MoveJ RelTool (starting_position, 124, 300, -195 \Rx:=-0.5, \Ry:=-1.8, \Rz:=0), v200, z200, Tooldata_7;
MoveJ RelTool (starting_position, 124, 300, -195 \Rx:=-0.2, \Ry:=-1.8, \Rz:=0), v200, z200, Tooldata_7;
MoveJ RelTool (starting_position, 124, 300, -195 \Rx:=0.2, \Ry:=-1.8, \Rz:=0), v200, z200, Tooldata_7;
MoveJ RelTool (starting_position, 125, 300, -194 \Rx:=0.6, \Ry:=-1.5, \Rz:=0), v200, z200, Tooldata_7;
MoveJ RelTool (starting_position, 125, 300, -194 \Rx:=1, \Ry:=-1.5, \Rz:=0), v200, z200, Tooldata_7;
MoveJ RelTool (starting_position, 126, 300, -193 \Rx:=1.5, \Ry:=-1.5, \Rz:=0), v200, z200, Tooldata_7;
MoveJ RelTool (starting_position, 127, 300, -193 \Rx:=2, \Ry:=-1.2, \Rz:=0), v200, z200, Tooldata_7;
MoveJ RelTool (starting_position, 128, 300, -192 \Rx:=2.5, \Ry:=-0.9, \Rz:=0), v200, z200, Tooldata_7;
MoveJ RelTool (starting_position, 130, 300, -192 \Rx:=3, \Ry:=-0.9, \Rz:=0), v200, z200, Tooldata_7;
MoveJ RelTool (starting_position, 132, 300, -191 \Rx:=3.4, \Ry:=-0.3, \Rz:=0), v200, z200, Tooldata_7;
MoveJ RelTool (starting_position, 134, 300, -191 \Rx:=3.9, \Ry:=0, \Rz:=0), v200, z200, Tooldata_7;
MoveJ RelTool (starting_position, 136, 300, -191 \Rx:=4.3, \Ry:=0.3, \Rz:=0), v200, z200, Tooldata_7;
MoveJ RelTool (starting_position, 138, 300, -190 \Rx:=4.6, \Ry:=0.6, \Rz:=0), v200, z200, Tooldata_7;
MoveJ RelTool (starting_position, 140, 300, -190 \Rx:=5, \Ry:=1.2, \Rz:=0), v200, z200, Tooldata_7;
MoveJ RelTool (starting_position, 143, 300, -189 \Rx:=5.3, \Ry:=1.5, \Rz:=0), v200, z200, Tooldata_7;
MoveJ RelTool (starting_position, 145, 300, -189 \Rx:=5.5, \Ry:=2.1, \Rz:=0), v200, z200, Tooldata_7;
MoveJ RelTool (starting_position, 148, 300, -189 \Rx:=5.7, \Ry:=2.4, \Rz:=0), v200, z200, Tooldata_7;
MoveJ RelTool (starting_position, 151, 300, -189 \Rx:=5.9, \Ry:=3, \Rz:=0), v200, z200, Tooldata_7;
MoveJ RelTool (starting_position, 155, 300, -189 \Rx:=6, \Ry:=3.6, \Rz:=0), v200, z200, Tooldata_7;
MoveJ RelTool (starting_position, 158, 300, -189 \Rx:=6.1, \Ry:=4.2, \Rz:=0), v200, z200, Tooldata_7;
MoveJ RelTool (starting_position, 162, 300, -189 \Rx:=6, \Ry:=4.8, \Rz:=0), v200, z200, Tooldata_7;
MoveJ RelTool (starting_position, 166, 300, -190 \Rx:=6, \Ry:=5.4, \Rz:=0), v200, z200, Tooldata_7;
MoveJ RelTool (starting_position, 170, 300, -190 \Rx:=5.9, \Ry:=6.3, \Rz:=0), v200, z200, Tooldata_7;
MoveJ RelTool (starting_position, 174, 300, -191 \Rx:=5.8, \Ry:=6.9, \Rz:=0), v200, z200, Tooldata_7;
MoveJ RelTool (starting_position, 178, 300, -191 \Rx:=5.7, \Ry:=7.8, \Rz:=0), v200, z200, Tooldata_7;
MoveJ RelTool (starting_position, 182, 300, -192 \Rx:=5.6, \Ry:=8.4, \Rz:=0), v200, z200, Tooldata_7;
MoveJ RelTool (starting_position, 186, 300, -193 \Rx:=5.5, \Ry:=9, \Rz:=0), v200, z200, Tooldata_7;
MoveJ RelTool (starting_position, 189, 300, -194 \Rx:=5.3, \Ry:=9.6, \Rz:=0), v200, z200, Tooldata_7;
MoveJ RelTool (starting_position, 193, 300, -195 \Rx:=5.3, \Ry:=10.5, \Rz:=0), v200, z200, Tooldata_7;
MoveJ RelTool (starting_position, 197, 300, -196 \Rx:=5.2, \Ry:=10.8, \Rz:=0), v200, z200, Tooldata_7;
MoveJ RelTool (starting_position, 200, 300, -197 \Rx:=5.2, \Ry:=11.7, \Rz:=0), v200, z200, Tooldata_7;
MoveJ RelTool (starting_position, 204, 300, -198 \Rx:=5.2, \Ry:=12.3, \Rz:=0), v200, z200, Tooldata_7;
MoveJ RelTool (starting_position, 207, 300, -199 \Rx:=5.3, \Ry:=12.6, \Rz:=0), v200, z200, Tooldata_7;
MoveJ RelTool (starting_position, 211, 300, -200 \Rx:=5.4, \Ry:=13.2, \Rz:=0), v200, z200, Tooldata_7;
MoveJ RelTool (starting_position, 214, 300, -202 \Rx:=5.5, \Ry:=14.1, \Rz:=0), v200, z200, Tooldata_7;
MoveJ RelTool (starting_position, 218, 300, -203 \Rx:=5.8, \Ry:=14.7, \Rz:=0), v200, z200, Tooldata_7;
MoveJ RelTool (starting_position, 221, 300, -205 \Rx:=5.9, \Ry:=15.3, \Rz:=0), v200, z200, Tooldata_7;
MoveJ RelTool (starting_position, 224, 300, -206 \Rx:=6.1, \Ry:=15.6, \Rz:=0), v200, z200, Tooldata_7;
MoveJ RelTool (starting_position, 227, 300, -208 \Rx:=6.4, \Ry:=16.2, \Rz:=0), v200, z200, Tooldata_7;
MoveJ RelTool (starting_position, 229, 300, -210 \Rx:=6.8, \Ry:=16.5, \Rz:=0), v200, z200, Tooldata_7;
MoveJ RelTool (starting_position, 231, 300, -212 \Rx:=7.2, \Ry:=17.1, \Rz:=0), v200, z200, Tooldata_7;
MoveJ RelTool (starting_position, 233, 300, -214 \Rx:=7.6, \Ry:=17.4, \Rz:=0), v200, z200, Tooldata_7;
MoveJ RelTool (starting_position, 235, 300, -216 \Rx:=8.1, \Ry:=17.7, \Rz:=0), v200, z200, Tooldata_7;
MoveJ RelTool (starting_position, 237, 300, -218 \Rx:=8.5, \Ry:=18, \Rz:=0), v200, z200, Tooldata_7;
MoveJ RelTool (starting_position, 238, 300, -221 \Rx:=8.9, \Ry:=18, \Rz:=0), v200, z200, Tooldata_7;
MoveJ RelTool (starting_position, 238, 300, -223 \Rx:=9.3, \Ry:=18.3, \Rz:=0), v200, z200, Tooldata_7;
MoveJ RelTool (starting_position, 238, 300, -226 \Rx:=9.8, \Ry:=18.3, \Rz:=0), v200, z200, Tooldata_7;
MoveJ RelTool (starting_position, 238, 300, -228 \Rx:=10.2, \Ry:=18.3, \Rz:=0), v200, z200, Tooldata_7;
MoveJ RelTool (starting_position, 238, 300, -231 \Rx:=10.5, \Ry:=18, \Rz:=0), v200, z200, Tooldata_7;
MoveJ RelTool (starting_position, 237, 300, -234 \Rx:=10.9, \Ry:=18, \Rz:=0), v200, z200, Tooldata_7;
MoveJ RelTool (starting_position, 235, 300, -237 \Rx:=11.2, \Ry:=17.7, \Rz:=0), v200, z200, Tooldata_7;
MoveJ RelTool (starting_position, 233, 300, -240 \Rx:=11.4, \Ry:=17.4, \Rz:=0), v200, z200, Tooldata_7;
MoveJ RelTool (starting_position, 231, 300, -243 \Rx:=11.6, \Ry:=17.1, \Rz:=0), v200, z200, Tooldata_7;
MoveJ RelTool (starting_position, 228, 300, -246 \Rx:=11.8, \Ry:=16.5, \Rz:=0), v200, z200, Tooldata_7;
MoveJ RelTool (starting_position, 225, 300, -249 \Rx:=12, \Ry:=15.9, \Rz:=0), v200, z200, Tooldata_7;
MoveJ RelTool (starting_position, 221, 300, -252 \Rx:=12.1, \Ry:=15.3, \Rz:=0), v200, z200, Tooldata_7;
MoveJ RelTool (starting_position, 216, 300, -255 \Rx:=12.2, \Ry:=14.4, \Rz:=0), v200, z200, Tooldata_7;
MoveJ RelTool (starting_position, 211, 300, -258 \Rx:=12.3, \Ry:=13.5, \Rz:=0), v200, z200, Tooldata_7;
MoveJ RelTool (starting_position, 206, 300, -261 \Rx:=12.4, \Ry:=12.6, \Rz:=0), v200, z200, Tooldata_7;
MoveJ RelTool (starting_position, 200, 300, -264 \Rx:=12.5, \Ry:=11.4, \Rz:=0), v200, z200, Tooldata_7;
MoveJ RelTool (starting_position, 194, 300, -266 \Rx:=12.6, \Ry:=10.5, \Rz:=0), v200, z200, Tooldata_7;
MoveJ RelTool (starting_position, 188, 300, -268 \Rx:=12.7, \Ry:=9.3, \Rz:=0), v200, z200, Tooldata_7;
MoveJ RelTool (starting_position, 181, 300, -270 \Rx:=12.8, \Ry:=8.4, \Rz:=0), v200, z200, Tooldata_7;
MoveJ RelTool (starting_position, 174, 300, -272 \Rx:=12.8, \Ry:=7.2, \Rz:=0), v200, z200, Tooldata_7;
MoveJ RelTool (starting_position, 167, 300, -273 \Rx:=12.9, \Ry:=5.7, \Rz:=0), v200, z200, Tooldata_7;
MoveJ RelTool (starting_position, 160, 300, -274 \Rx:=13, \Ry:=4.5, \Rz:=0), v200, z200, Tooldata_7;
MoveJ RelTool (starting_position, 153, 300, -275 \Rx:=13.1, \Ry:=3.3, \Rz:=0), v200, z200, Tooldata_7;
MoveJ RelTool (starting_position, 146, 300, -276 \Rx:=13.1, \Ry:=2.1, \Rz:=0), v200, z200, Tooldata_7;
MoveJ RelTool (starting_position, 138, 300, -276 \Rx:=13.2, \Ry:=0.6, \Rz:=0), v200, z200, Tooldata_7;
MoveJ RelTool (starting_position, 131, 300, -276 \Rx:=13.3, \Ry:=-0.6, \Rz:=0), v200, z200, Tooldata_7;
MoveJ RelTool (starting_position, 124, 300, -275 \Rx:=13.4, \Ry:=-1.8, \Rz:=0), v200, z200, Tooldata_7;
MoveJ RelTool (starting_position, 117, 300, -275 \Rx:=13.5, \Ry:=-3, \Rz:=0), v200, z200, Tooldata_7;
MoveJ RelTool (starting_position, 110, 300, -274 \Rx:=13.5, \Ry:=-4.2, \Rz:=0), v200, z200, Tooldata_7;
MoveJ RelTool (starting_position, 104, 300, -273 \Rx:=13.6, \Ry:=-5.4, \Rz:=0), v200, z200, Tooldata_7;
MoveJ RelTool (starting_position, 97, 300, -271 \Rx:=13.7, \Ry:=-6.3, \Rz:=0), v200, z200, Tooldata_7;
MoveJ RelTool (starting_position, 91, 300, -270 \Rx:=13.7, \Ry:=-7.5, \Rz:=0), v200, z200, Tooldata_7;
MoveJ RelTool (starting_position, 85, 300, -268 \Rx:=13.8, \Ry:=-8.4, \Rz:=0), v200, z200, Tooldata_7;
MoveJ RelTool (starting_position, 80, 300, -266 \Rx:=13.8, \Ry:=-9.6, \Rz:=0), v200, z200, Tooldata_7;
MoveJ RelTool (starting_position, 75, 300, -264 \Rx:=13.9, \Ry:=-10.5, \Rz:=0), v200, z200, Tooldata_7;
MoveJ RelTool (starting_position, 70, 300, -262 \Rx:=13.9, \Ry:=-11.1, \Rz:=0), v200, z200, Tooldata_7;
MoveJ RelTool (starting_position, 65, 300, -260 \Rx:=14, \Ry:=-12, \Rz:=0), v200, z200, Tooldata_7;
MoveJ RelTool (starting_position, 61, 300, -258 \Rx:=14.1, \Ry:=-12.9, \Rz:=0), v200, z200, Tooldata_7;
MoveJ RelTool (starting_position, 57, 300, -256 \Rx:=14.1, \Ry:=-13.5, \Rz:=0), v200, z200, Tooldata_7;
MoveJ RelTool (starting_position, 54, 300, -253 \Rx:=14.2, \Ry:=-14.1, \Rz:=0), v200, z200, Tooldata_7;
MoveJ RelTool (starting_position, 51, 300, -251 \Rx:=14.3, \Ry:=-14.4, \Rz:=0), v200, z200, Tooldata_7;
MoveJ RelTool (starting_position, 48, 300, -249 \Rx:=14.3, \Ry:=-15, \Rz:=0), v200, z200, Tooldata_7;
MoveJ RelTool (starting_position, 46, 300, -246 \Rx:=14.4, \Ry:=-15.3, \Rz:=0), v200, z200, Tooldata_7;
MoveJ RelTool (starting_position, 44, 300, -244 \Rx:=14.5, \Ry:=-15.6, \Rz:=0), v200, z200, Tooldata_7;
MoveJ RelTool (starting_position, 42, 300, -242 \Rx:=14.6, \Ry:=-15.9, \Rz:=0), v200, z200, Tooldata_7;
MoveJ RelTool (starting_position, 41, 300, -240 \Rx:=14.6, \Ry:=-16.2, \Rz:=0), v200, z200, Tooldata_7;
MoveJ RelTool (starting_position, 39, 300, -238 \Rx:=14.6, \Ry:=-16.5, \Rz:=0), v200, z200, Tooldata_7;
MoveJ RelTool (starting_position, 38, 300, -236 \Rx:=14.6, \Ry:=-16.5, \Rz:=0), v200, z200, Tooldata_7;
MoveJ RelTool (starting_position, 37, 300, -234 \Rx:=14.7, \Ry:=-16.8, \Rz:=0), v200, z200, Tooldata_7;
MoveJ RelTool (starting_position, 37, 300, -232 \Rx:=14.6, \Ry:=-16.8, \Rz:=0), v200, z200, Tooldata_7;
MoveJ RelTool (starting_position, 36, 300, -230 \Rx:=14.6, \Ry:=-17.1, \Rz:=0), v200, z200, Tooldata_7;
MoveJ RelTool (starting_position, 35, 300, -228 \Rx:=14.6, \Ry:=-17.1, \Rz:=0), v200, z200, Tooldata_7;
MoveJ RelTool (starting_position, 35, 300, -227 \Rx:=14.6, \Ry:=-17.1, \Rz:=0), v200, z200, Tooldata_7;
MoveJ RelTool (starting_position, 34, 300, -225 \Rx:=14.6, \Ry:=-17.1, \Rz:=0), v200, z200, Tooldata_7;
MoveJ RelTool (starting_position, 34, 300, -224 \Rx:=14.5, \Ry:=-17.4, \Rz:=0), v200, z200, Tooldata_7;
MoveJ RelTool (starting_position, 33, 300, -222 \Rx:=14.4, \Ry:=-17.4, \Rz:=0), v200, z200, Tooldata_7;
MoveJ RelTool (starting_position, 33, 300, -221 \Rx:=14.3, \Ry:=-17.4, \Rz:=0), v200, z200, Tooldata_7;
MoveJ RelTool (starting_position, 32, 300, -219 \Rx:=14.2, \Ry:=-17.7, \Rz:=0), v200, z200, Tooldata_7;
MoveJ RelTool (starting_position, 32, 300, -218 \Rx:=14.1, \Ry:=-17.7, \Rz:=0), v200, z200, Tooldata_7;
MoveJ RelTool (starting_position, 31, 300, -216 \Rx:=13.9, \Ry:=-17.7, \Rz:=0), v200, z200, Tooldata_7;
MoveJ RelTool (starting_position, 30, 300, -215 \Rx:=13.7, \Ry:=-18, \Rz:=0), v200, z200, Tooldata_7;
MoveJ RelTool (starting_position, 30, 300, -214 \Rx:=13.5, \Ry:=-18, \Rz:=0), v200, z200, Tooldata_7;
MoveJ RelTool (starting_position, 29, 300, -212 \Rx:=13.3, \Ry:=-18, \Rz:=0), v200, z200, Tooldata_7;
MoveJ RelTool (starting_position, 28, 300, -211 \Rx:=13.1, \Ry:=-18.3, \Rz:=0), v200, z200, Tooldata_7;
MoveJ RelTool (starting_position, 27, 300, -209 \Rx:=12.8, \Ry:=-18.3, \Rz:=0), v200, z200, Tooldata_7;
MoveJ RelTool (starting_position, 26, 300, -208 \Rx:=12.5, \Ry:=-18.6, \Rz:=0), v200, z200, Tooldata_7;
MoveJ RelTool (starting_position, 25, 300, -206 \Rx:=12.1, \Ry:=-18.9, \Rz:=0), v200, z200, Tooldata_7;
MoveJ RelTool (starting_position, 24, 300, -204 \Rx:=11.7, \Ry:=-19.2, \Rz:=0), v200, z200, Tooldata_7;
MoveJ RelTool (starting_position, 23, 300, -203 \Rx:=11.2, \Ry:=-19.2, \Rz:=0), v200, z200, Tooldata_7;
MoveJ RelTool (starting_position, 22, 300, -201 \Rx:=10.7, \Ry:=-19.5, \Rz:=0), v200, z200, Tooldata_7;
MoveJ RelTool (starting_position, 21, 300, -199 \Rx:=10.2, \Ry:=-19.5, \Rz:=0), v200, z200, Tooldata_7;
MoveJ RelTool (starting_position, 20, 300, -197 \Rx:=9.5, \Ry:=-19.5, \Rz:=0), v200, z200, Tooldata_7;
MoveJ RelTool (starting_position, 18, 300, -195 \Rx:=8.8, \Ry:=-20.1, \Rz:=0), v200, z200, Tooldata_7;
MoveJ RelTool (starting_position, 17, 300, -193 \Rx:=8.1, \Ry:=-20.4, \Rz:=0), v200, z200, Tooldata_7;
MoveJ RelTool (starting_position, 16, 300, -191 \Rx:=7.3, \Ry:=-20.4, \Rz:=0), v200, z200, Tooldata_7;
MoveJ RelTool (starting_position, 15, 300, -188 \Rx:=6.6, \Ry:=-20.7, \Rz:=0), v200, z200, Tooldata_7;
MoveJ RelTool (starting_position, 14, 300, -186 \Rx:=5.7, \Ry:=-20.7, \Rz:=0), v200, z200, Tooldata_7;
MoveJ RelTool (starting_position, 13, 300, -183 \Rx:=4.8, \Ry:=-21, \Rz:=0), v200, z200, Tooldata_7;
MoveJ RelTool (starting_position, 13, 300, -181 \Rx:=3.9, \Ry:=-21, \Rz:=0), v200, z200, Tooldata_7;
MoveJ RelTool (starting_position, 12, 300, -178 \Rx:=2.9, \Ry:=-21, \Rz:=0), v200, z200, Tooldata_7;
MoveJ RelTool (starting_position, 11, 300, -176 \Rx:=2, \Ry:=-21.3, \Rz:=0), v200, z200, Tooldata_7;
MoveJ RelTool (starting_position, 11, 300, -173 \Rx:=1.1, \Ry:=-21.3, \Rz:=0), v200, z200, Tooldata_7;
MoveJ RelTool (starting_position, 10, 300, -170 \Rx:=0.2, \Ry:=-21.6, \Rz:=0), v200, z200, Tooldata_7;
MoveJ RelTool (starting_position, 10, 300, -167 \Rx:=-0.7, \Ry:=-21.6, \Rz:=0), v200, z200, Tooldata_7;
MoveJ RelTool (starting_position, 10, 300, -164 \Rx:=-1.4, \Ry:=-21.6, \Rz:=0), v200, z200, Tooldata_7;
MoveJ RelTool (starting_position, 11, 300, -162 \Rx:=-2.1, \Ry:=-21.3, \Rz:=0), v200, z200, Tooldata_7;
MoveJ RelTool (starting_position, 12, 300, -159 \Rx:=-2.8, \Ry:=-21, \Rz:=0), v200, z200, Tooldata_7;
MoveJ RelTool (starting_position, 14, 300, -156 \Rx:=-3.3, \Ry:=-20.7, \Rz:=0), v200, z200, Tooldata_7;
MoveJ RelTool (starting_position, 15, 300, -153 \Rx:=-3.7, \Ry:=-20.7, \Rz:=0), v200, z200, Tooldata_7;
MoveJ RelTool (starting_position, 17, 300, -151 \Rx:=-4, \Ry:=-20.4, \Rz:=0), v200, z200, Tooldata_7;
MoveJ RelTool (starting_position, 18, 300, -148 \Rx:=-4.2, \Ry:=-20.1, \Rz:=0), v200, z200, Tooldata_7;
MoveJ RelTool (starting_position, 21, 300, -146 \Rx:=-4.3, \Ry:=-19.8, \Rz:=0), v200, z200, Tooldata_7;
MoveJ RelTool (starting_position, 23, 300, -144 \Rx:=-4.2, \Ry:=-19.2, \Rz:=0), v200, z200, Tooldata_7;
MoveJ RelTool (starting_position, 25, 300, -141 \Rx:=-3.9, \Ry:=-18.6, \Rz:=0), v200, z200, Tooldata_7;
MoveJ RelTool (starting_position, 28, 300, -139 \Rx:=-3.7, \Ry:=-18.3, \Rz:=0), v200, z200, Tooldata_7;
MoveJ RelTool (starting_position, 30, 300, -137 \Rx:=-3.3, \Ry:=-18, \Rz:=0), v200, z200, Tooldata_7;
MoveJ RelTool (starting_position, 32, 300, -136 \Rx:=-2.8, \Ry:=-17.4, \Rz:=0), v200, z200, Tooldata_7;
MoveJ RelTool (starting_position, 34, 300, -134 \Rx:=-2.2, \Ry:=-17.4, \Rz:=0), v200, z200, Tooldata_7;
MoveJ RelTool (starting_position, 37, 300, -133 \Rx:=-1.5, \Ry:=-17.1, \Rz:=0), v200, z200, Tooldata_7;
MoveJ RelTool (starting_position, 40, 300, -132 \Rx:=-0.8, \Ry:=-16.2, \Rz:=0), v200, z200, Tooldata_7;
MoveJ RelTool (starting_position, 44, 300, -131 \Rx:=0, \Ry:=-15.6, \Rz:=0), v200, z200, Tooldata_7;
MoveJ RelTool (starting_position, 47, 300, -131 \Rx:=0.9, \Ry:=-15, \Rz:=0), v200, z200, Tooldata_7;
MoveJ RelTool (starting_position, 51, 300, -130 \Rx:=1.7, \Ry:=-14.4, \Rz:=0), v200, z200, Tooldata_7;
MoveJ RelTool (starting_position, 55, 300, -130 \Rx:=2.4, \Ry:=-13.5, \Rz:=0), v200, z200, Tooldata_7;
MoveJ RelTool (starting_position, 59, 300, -131 \Rx:=3.2, \Ry:=-12.9, \Rz:=0), v200, z200, Tooldata_7;
MoveJ RelTool (starting_position, 63, 300, -131 \Rx:=3.9, \Ry:=-12, \Rz:=0), v200, z200, Tooldata_7;
MoveJ RelTool (starting_position, 67, 299.9, -131 \Rx:=4.6, \Ry:=-11.4, \Rz:=0), v200, z200, Tooldata_7;
MoveJ RelTool (starting_position, 70, 299.9, -132 \Rx:=5.3, \Ry:=-10.8, \Rz:=0), v200, z200, Tooldata_7;
MoveJ RelTool (starting_position, 73, 299.8, -133 \Rx:=5.8, \Ry:=-10.5, \Rz:=0), v200, z200, Tooldata_7;
MoveJ RelTool (starting_position, 76, 299.7, -134 \Rx:=6.2, \Ry:=-9.9, \Rz:=0), v200, z200, Tooldata_7;
MoveJ RelTool (starting_position, 78, 299.7, -135 \Rx:=6.6, \Ry:=-9.6, \Rz:=0), v200, z200, Tooldata_7;
MoveJ RelTool (starting_position, 81, 299.6, -136 \Rx:=6.9, \Ry:=-9.3, \Rz:=0), v200, z200, Tooldata_7;
MoveJ RelTool (starting_position, 84, 299.5, -137 \Rx:=7.1, \Ry:=-8.7, \Rz:=0), v200, z200, Tooldata_7;
MoveJ RelTool (starting_position, 87, 299.3, -138 \Rx:=7.3, \Ry:=-8.1, \Rz:=0), v200, z200, Tooldata_7;
MoveJ RelTool (starting_position, 90, 299.2, -138 \Rx:=7.4, \Ry:=-7.5, \Rz:=0), v200, z200, Tooldata_7;
MoveJ RelTool (starting_position, 93, 299.1, -139 \Rx:=7.4, \Ry:=-6.9, \Rz:=0), v200, z200, Tooldata_7;
MoveJ RelTool (starting_position, 95, 298.9, -139 \Rx:=7.2, \Ry:=-6.6, \Rz:=0), v200, z200, Tooldata_7;
MoveJ RelTool (starting_position, 98, 298.7, -139 \Rx:=7, \Ry:=-6, \Rz:=0), v200, z200, Tooldata_7;
MoveJ RelTool (starting_position, 100, 298.5, -139 \Rx:=6.8, \Ry:=-5.7, \Rz:=0), v200, z200, Tooldata_7;
MoveJ RelTool (starting_position, 102, 298.3, -138 \Rx:=6.6, \Ry:=-5.7, \Rz:=0), v200, z200, Tooldata_7;
MoveJ RelTool (starting_position, 105, 298.1, -138 \Rx:=6.3, \Ry:=-5.1, \Rz:=0), v200, z200, Tooldata_7;
MoveJ RelTool (starting_position, 107, 297.8, -137 \Rx:=6, \Ry:=-4.5, \Rz:=0), v200, z200, Tooldata_7;
MoveJ RelTool (starting_position, 110, 297.5, -136 \Rx:=5.6, \Ry:=-4.2, \Rz:=0), v200, z200, Tooldata_7;
MoveJ RelTool (starting_position, 113, 297.2, -134 \Rx:=5.2, \Ry:=-3.6, \Rz:=0), v200, z200, Tooldata_7;
MoveJ RelTool (starting_position, 115, 296.8, -133 \Rx:=4.9, \Ry:=-3.3, \Rz:=0), v200, z200, Tooldata_7;
MoveJ RelTool (starting_position, 118, 296.4, -131 \Rx:=4.4, \Ry:=-2.7, \Rz:=0), v200, z200, Tooldata_7;
MoveJ RelTool (starting_position, 121, 296, -129 \Rx:=4.1, \Ry:=-2.1, \Rz:=0), v200, z200, Tooldata_7;
MoveJ RelTool (starting_position, 124, 295.6, -126 \Rx:=3.7, \Ry:=-1.8, \Rz:=0), v200, z200, Tooldata_7;
MoveJ RelTool (starting_position, 127, 295.2, -123 \Rx:=3.4, \Ry:=-1.2, \Rz:=0), v200, z200, Tooldata_7;
MoveJ RelTool (starting_position, 130, 294.7, -121 \Rx:=3, \Ry:=-0.6, \Rz:=0), v200, z200, Tooldata_7;
MoveJ RelTool (starting_position, 133, 294.1, -118 \Rx:=2.6, \Ry:=-0, \Rz:=0), v200, z200, Tooldata_7;
MoveJ RelTool (starting_position, 137, 293.6, -115 \Rx:=2.3, \Ry:=0.6, \Rz:=0), v200, z200, Tooldata_7;
MoveJ RelTool (starting_position, 140, 293, -112 \Rx:=2, \Ry:=0.9, \Rz:=0), v200, z200, Tooldata_7;
MoveJ RelTool (starting_position, 144, 292.4, -109 \Rx:=1.7, \Ry:=1.8, \Rz:=0), v200, z200, Tooldata_7;
MoveJ RelTool (starting_position, 147, 291.8, -107 \Rx:=1.4, \Ry:=2.4, \Rz:=0), v200, z200, Tooldata_7;
MoveJ RelTool (starting_position, 151, 291.2, -104 \Rx:=1.1, \Ry:=3, \Rz:=0), v200, z200, Tooldata_7;
MoveJ RelTool (starting_position, 154, 290.5, -101 \Rx:=0.8, \Ry:=3.6, \Rz:=0), v200, z200, Tooldata_7;
MoveJ RelTool (starting_position, 158, 289.8, -98 \Rx:=0.6, \Ry:=4.2, \Rz:=0), v200, z200, Tooldata_7;
MoveJ RelTool (starting_position, 162, 289.1, -96 \Rx:=0.3, \Ry:=4.8, \Rz:=0), v200, z200, Tooldata_7;
MoveJ RelTool (starting_position, 165, 288.4, -94 \Rx:=0.1, \Ry:=5.4, \Rz:=0), v200, z200, Tooldata_7;
MoveJ RelTool (starting_position, 169, 287.6, -92 \Rx:=-0.1, \Ry:=6.3, \Rz:=0), v200, z200, Tooldata_7;
MoveJ RelTool (starting_position, 172, 286.9, -90 \Rx:=-0.3, \Ry:=6.6, \Rz:=0), v200, z200, Tooldata_7;
MoveJ RelTool (starting_position, 175, 286.2, -88 \Rx:=-0.5, \Ry:=7.2, \Rz:=0), v200, z200, Tooldata_7;
MoveJ RelTool (starting_position, 179, 285.4, -87 \Rx:=-0.6, \Ry:=7.8, \Rz:=0), v200, z200, Tooldata_7;
MoveJ RelTool (starting_position, 182, 284.6, -86 \Rx:=-0.6, \Ry:=8.4, \Rz:=0), v200, z200, Tooldata_7;
MoveJ RelTool (starting_position, 185, 283.9, -85 \Rx:=-0.6, \Ry:=9, \Rz:=0), v200, z200, Tooldata_7;
MoveJ RelTool (starting_position, 187, 283.1, -84 \Rx:=-0.6, \Ry:=9.6, \Rz:=0), v200, z200, Tooldata_7;
MoveJ RelTool (starting_position, 189, 282.4, -83 \Rx:=-0.6, \Ry:=9.9, \Rz:=0), v200, z200, Tooldata_7;
MoveJ RelTool (starting_position, 191, 281.7, -82 \Rx:=-0.5, \Ry:=9.9, \Rz:=0), v200, z200, Tooldata_7;
MoveJ RelTool (starting_position, 193, 280.9, -82 \Rx:=-0.3, \Ry:=10.2, \Rz:=0), v200, z200, Tooldata_7;
MoveJ RelTool (starting_position, 194, 280.2, -81 \Rx:=-0, \Ry:=10.5, \Rz:=0), v200, z200, Tooldata_7;
MoveJ RelTool (starting_position, 196, 279.5, -81 \Rx:=0.3, \Ry:=10.8, \Rz:=0), v200, z200, Tooldata_7;
MoveJ RelTool (starting_position, 198, 278.9, -81 \Rx:=0.7, \Ry:=11.1, \Rz:=0), v200, z200, Tooldata_7;
MoveJ RelTool (starting_position, 199, 278.2, -81 \Rx:=1.2, \Ry:=11.4, \Rz:=0), v200, z200, Tooldata_7;
MoveJ RelTool (starting_position, 201, 277.6, -81 \Rx:=1.7, \Ry:=11.7, \Rz:=0), v200, z200, Tooldata_7;
MoveJ RelTool (starting_position, 202, 277, -81 \Rx:=2.3, \Ry:=12, \Rz:=0), v200, z200, Tooldata_7;
MoveJ RelTool (starting_position, 202, 276.4, -82 \Rx:=2.9, \Ry:=12, \Rz:=0), v200, z200, Tooldata_7;
MoveJ RelTool (starting_position, 203, 275.9, -82 \Rx:=3.6, \Ry:=12, \Rz:=0), v200, z200, Tooldata_7;
MoveJ RelTool (starting_position, 203, 275.4, -83 \Rx:=4.3, \Ry:=12, \Rz:=0), v200, z200, Tooldata_7;
MoveJ RelTool (starting_position, 203, 274.9, -83 \Rx:=5, \Ry:=12, \Rz:=0), v200, z200, Tooldata_7;
MoveJ RelTool (starting_position, 202, 274.4, -84 \Rx:=5.8, \Ry:=12, \Rz:=0), v200, z200, Tooldata_7;
MoveJ RelTool (starting_position, 201, 274, -85 \Rx:=6.6, \Ry:=11.7, \Rz:=0), v200, z200, Tooldata_7;
MoveJ RelTool (starting_position, 200, 273.6, -87 \Rx:=7.3, \Ry:=11.7, \Rz:=0), v200, z200, Tooldata_7;
MoveJ RelTool (starting_position, 198, 273.2, -88 \Rx:=8.1, \Ry:=11.1, \Rz:=0), v200, z200, Tooldata_7;
MoveJ RelTool (starting_position, 196, 272.9, -90 \Rx:=8.9, \Ry:=10.8, \Rz:=0), v200, z200, Tooldata_7;
MoveJ RelTool (starting_position, 195, 272.5, -92 \Rx:=9.6, \Ry:=10.5, \Rz:=0), v200, z200, Tooldata_7;
MoveJ RelTool (starting_position, 193, 272.3, -93 \Rx:=10.4, \Ry:=10.2, \Rz:=0), v200, z200, Tooldata_7;
MoveJ RelTool (starting_position, 191, 272, -95 \Rx:=11.1, \Ry:=9.9, \Rz:=0), v200, z200, Tooldata_7;
MoveJ RelTool (starting_position, 188, 271.7, -96 \Rx:=11.8, \Ry:=9.6, \Rz:=0), v200, z200, Tooldata_7;
MoveJ RelTool (starting_position, 186, 271.5, -98 \Rx:=12.4, \Ry:=9.3, \Rz:=0), v200, z200, Tooldata_7;
MoveJ RelTool (starting_position, 183, 271.3, -99 \Rx:=13, \Ry:=8.7, \Rz:=0), v200, z200, Tooldata_7;
MoveJ RelTool (starting_position, 180, 271.1, -101 \Rx:=13.5, \Ry:=7.8, \Rz:=0), v200, z200, Tooldata_7;
MoveJ RelTool (starting_position, 176, 271, -102 \Rx:=14, \Ry:=7.2, \Rz:=0), v200, z200, Tooldata_7;
MoveJ RelTool (starting_position, 173, 270.8, -103 \Rx:=14.4, \Ry:=6.6, \Rz:=0), v200, z200, Tooldata_7;
MoveJ RelTool (starting_position, 171, 270.7, -104 \Rx:=14.8, \Ry:=6.3, \Rz:=0), v200, z200, Tooldata_7;
MoveJ RelTool (starting_position, 168, 270.6, -105 \Rx:=15.1, \Ry:=6, \Rz:=0), v200, z200, Tooldata_7;
MoveJ RelTool (starting_position, 165, 270.5, -106 \Rx:=15.4, \Ry:=5.7, \Rz:=0), v200, z200, Tooldata_7;
MoveJ RelTool (starting_position, 162, 270.4, -107 \Rx:=15.7, \Ry:=5.1, \Rz:=0), v200, z200, Tooldata_7;
MoveJ RelTool (starting_position, 159, 270.3, -108 \Rx:=15.9, \Ry:=4.5, \Rz:=0), v200, z200, Tooldata_7;
MoveJ RelTool (starting_position, 155, 270.2, -108 \Rx:=16, \Ry:=3.6, \Rz:=0), v200, z200, Tooldata_7;
MoveJ RelTool (starting_position, 151, 270.2, -108 \Rx:=16, \Ry:=3, \Rz:=0), v200, z200, Tooldata_7;
MoveJ RelTool (starting_position, 147, 270.1, -108 \Rx:=15.9, \Ry:=2.1, \Rz:=0), v200, z200, Tooldata_7;
MoveJ RelTool (starting_position, 143, 270.1, -108 \Rx:=15.8, \Ry:=1.2, \Rz:=0), v200, z200, Tooldata_7;
MoveJ RelTool (starting_position, 140, 270, -108 \Rx:=15.7, \Ry:=0.9, \Rz:=0), v200, z200, Tooldata_7;
MoveJ RelTool (starting_position, 137, 270, -108 \Rx:=15.5, \Ry:=0.3, \Rz:=0), v200, z200, Tooldata_7;
MoveJ RelTool (starting_position, 135, 270, -107 \Rx:=15.2, \Ry:=0, \Rz:=0), v200, z200, Tooldata_7;
MoveJ RelTool (starting_position, 134, 270, -107 \Rx:=14.8, \Ry:=-0, \Rz:=0), v200, z200, Tooldata_7;
MoveJ RelTool (starting_position, 134, 270, -106 \Rx:=14.4, \Ry:=-0.3, \Rz:=0), v200, z200, Tooldata_7;
MoveJ RelTool (starting_position, 134, 270, -105 \Rx:=14.1, \Ry:=-0, \Rz:=0), v200, z200, Tooldata_7;
MoveJ RelTool (starting_position, 134, 270, -104 \Rx:=13.6, \Ry:=-0, \Rz:=0), v200, z200, Tooldata_7;
MoveJ RelTool (starting_position, 134, 270, -104 \Rx:=13.1, \Ry:=0, \Rz:=0), v200, z200, Tooldata_7;
MoveJ RelTool (starting_position, 135, 270, -103 \Rx:=12.5, \Ry:=0.3, \Rz:=0), v200, z200, Tooldata_7;
MoveJ RelTool (starting_position, 136, 270, -102 \Rx:=11.9, \Ry:=0.3, \Rz:=0), v200, z200, Tooldata_7;
MoveJ RelTool (starting_position, 137, 270, -102 \Rx:=11.3, \Ry:=0.6, \Rz:=0), v200, z200, Tooldata_7;
MoveJ RelTool (starting_position, 138, 270, -102 \Rx:=10.5, \Ry:=0.6, \Rz:=0), v200, z200, Tooldata_7;
MoveJ RelTool (starting_position, 140, 270, -101 \Rx:=9.9, \Ry:=0.9, \Rz:=0), v200, z200, Tooldata_7;
MoveJ RelTool (starting_position, 142, 270, -101 \Rx:=9.1, \Ry:=1.5, \Rz:=0), v200, z200, Tooldata_7;
MoveJ RelTool (starting_position, 145, 270, -101 \Rx:=8.3, \Ry:=1.8, \Rz:=0), v200, z200, Tooldata_7;
MoveJ RelTool (starting_position, 147, 270, -101 \Rx:=7.5, \Ry:=2.4, \Rz:=0), v200, z200, Tooldata_7;
MoveJ RelTool (starting_position, 150, 270, -101 \Rx:=6.7, \Ry:=3, \Rz:=0), v200, z200, Tooldata_7;
MoveJ RelTool (starting_position, 152, 270, -101 \Rx:=6, \Ry:=3, \Rz:=0), v200, z200, Tooldata_7;
MoveJ RelTool (starting_position, 155, 270, -102 \Rx:=5.2, \Ry:=3.6, \Rz:=0), v200, z200, Tooldata_7;
MoveJ RelTool (starting_position, 159, 270, -103 \Rx:=4.5, \Ry:=4.2, \Rz:=0), v200, z200, Tooldata_7;
MoveJ RelTool (starting_position, 162, 270, -104 \Rx:=3.7, \Ry:=4.8, \Rz:=0), v200, z200, Tooldata_7;
MoveJ RelTool (starting_position, 167, 270, -106 \Rx:=3.1, \Ry:=5.7, \Rz:=0), v200, z200, Tooldata_7;
MoveJ RelTool (starting_position, 171, 270, -107 \Rx:=2.4, \Ry:=6.6, \Rz:=0), v200, z200, Tooldata_7;
MoveJ RelTool (starting_position, 175, 270, -109 \Rx:=1.8, \Ry:=7.2, \Rz:=0), v200, z200, Tooldata_7;
MoveJ RelTool (starting_position, 179, 270, -111 \Rx:=1.2, \Ry:=7.8, \Rz:=0), v200, z200, Tooldata_7;
MoveJ RelTool (starting_position, 184, 270, -113 \Rx:=0.7, \Ry:=8.7, \Rz:=0), v200, z200, Tooldata_7;
MoveJ RelTool (starting_position, 188, 270, -116 \Rx:=0.1, \Ry:=9.6, \Rz:=0), v200, z200, Tooldata_7;
MoveJ RelTool (starting_position, 192, 270, -118 \Rx:=-0.3, \Ry:=10.2, \Rz:=0), v200, z200, Tooldata_7;
MoveJ RelTool (starting_position, 196, 270, -121 \Rx:=-0.7, \Ry:=10.8, \Rz:=0), v200, z200, Tooldata_7;
MoveJ RelTool (starting_position, 199, 270, -124 \Rx:=-1.1, \Ry:=11.4, \Rz:=0), v200, z200, Tooldata_7;
MoveJ RelTool (starting_position, 202, 270, -128 \Rx:=-1.5, \Ry:=12, \Rz:=0), v200, z200, Tooldata_7;
MoveJ RelTool (starting_position, 205, 270, -131 \Rx:=-1.9, \Ry:=12.3, \Rz:=0), v200, z200, Tooldata_7;
MoveJ RelTool (starting_position, 208, 270, -135 \Rx:=-2.2, \Ry:=12.9, \Rz:=0), v200, z200, Tooldata_7;
MoveJ RelTool (starting_position, 211, 270, -139 \Rx:=-2.6, \Ry:=13.5, \Rz:=0), v200, z200, Tooldata_7;
MoveJ RelTool (starting_position, 214, 270, -143 \Rx:=-2.9, \Ry:=14.1, \Rz:=0), v200, z200, Tooldata_7;
MoveJ RelTool (starting_position, 217, 270, -147 \Rx:=-3.2, \Ry:=14.7, \Rz:=0), v200, z200, Tooldata_7;
MoveJ RelTool (starting_position, 219, 270, -151 \Rx:=-3.6, \Ry:=15, \Rz:=0), v200, z200, Tooldata_7;
MoveJ RelTool (starting_position, 220, 270, -156 \Rx:=-3.9, \Ry:=15, \Rz:=0), v200, z200, Tooldata_7;
MoveJ RelTool (starting_position, 222, 270, -160 \Rx:=-4.1, \Ry:=15.3, \Rz:=0), v200, z200, Tooldata_7;
MoveJ RelTool (starting_position, 223, 270, -165 \Rx:=-4.3, \Ry:=15.3, \Rz:=0), v200, z200, Tooldata_7;
MoveJ RelTool (starting_position, 224, 270, -170 \Rx:=-4.5, \Ry:=15.6, \Rz:=0), v200, z200, Tooldata_7;
MoveJ RelTool (starting_position, 225, 270, -175 \Rx:=-4.7, \Ry:=15.9, \Rz:=0), v200, z200, Tooldata_7;
MoveJ RelTool (starting_position, 225, 270, -180 \Rx:=-4.8, \Ry:=16.2, \Rz:=0), v200, z200, Tooldata_7;
MoveJ RelTool (starting_position, 226, 270, -185 \Rx:=-4.9, \Ry:=16.2, \Rz:=0), v200, z200, Tooldata_7;
MoveJ RelTool (starting_position, 225, 270, -190 \Rx:=-4.9, \Ry:=15.9, \Rz:=0), v200, z200, Tooldata_7;
MoveJ RelTool (starting_position, 224, 270, -195 \Rx:=-4.9, \Ry:=15.6, \Rz:=0), v200, z200, Tooldata_7;
MoveJ RelTool (starting_position, 223, 270, -200 \Rx:=-4.7, \Ry:=15.6, \Rz:=0), v200, z200, Tooldata_7;
MoveJ RelTool (starting_position, 221, 270, -204 \Rx:=-4.6, \Ry:=15.3, \Rz:=0), v200, z200, Tooldata_7;
MoveJ RelTool (starting_position, 219, 270, -208 \Rx:=-4.4, \Ry:=15, \Rz:=0), v200, z200, Tooldata_7;
MoveJ RelTool (starting_position, 217, 270, -212 \Rx:=-4.3, \Ry:=14.7, \Rz:=0), v200, z200, Tooldata_7;
MoveJ RelTool (starting_position, 214, 270, -215 \Rx:=-4.2, \Ry:=14.1, \Rz:=0), v200, z200, Tooldata_7;
MoveJ RelTool (starting_position, 210, 270, -218 \Rx:=-4, \Ry:=13.2, \Rz:=0), v200, z200, Tooldata_7;
MoveJ RelTool (starting_position, 206, 270, -221 \Rx:=-3.7, \Ry:=12.6, \Rz:=0), v200, z200, Tooldata_7;
MoveJ RelTool (starting_position, 201, 270, -223 \Rx:=-3.5, \Ry:=11.7, \Rz:=0), v200, z200, Tooldata_7;
MoveJ RelTool (starting_position, 197, 270, -225 \Rx:=-3.3, \Ry:=10.8, \Rz:=0), v200, z200, Tooldata_7;
MoveJ RelTool (starting_position, 192, 270, -226 \Rx:=-3.2, \Ry:=10.2, \Rz:=0), v200, z200, Tooldata_7;
MoveJ RelTool (starting_position, 187, 270, -227 \Rx:=-3.1, \Ry:=9.3, \Rz:=0), v200, z200, Tooldata_7;
MoveJ RelTool (starting_position, 182, 270, -228 \Rx:=-3, \Ry:=8.4, \Rz:=0), v200, z200, Tooldata_7;
MoveJ RelTool (starting_position, 177, 270, -228 \Rx:=-2.9, \Ry:=7.5, \Rz:=0), v200, z200, Tooldata_7;
MoveJ RelTool (starting_position, 172, 270, -227 \Rx:=-2.9, \Ry:=6.6, \Rz:=0), v200, z200, Tooldata_7;
MoveJ RelTool (starting_position, 167, 270, -227 \Rx:=-2.8, \Ry:=6, \Rz:=0), v200, z200, Tooldata_7;
MoveJ RelTool (starting_position, 162, 270, -226 \Rx:=-2.8, \Ry:=4.8, \Rz:=0), v200, z200, Tooldata_7;
MoveJ RelTool (starting_position, 156, 270, -225 \Rx:=-2.7, \Ry:=3.9, \Rz:=0), v200, z200, Tooldata_7;
MoveJ RelTool (starting_position, 151, 270, -223 \Rx:=-2.6, \Ry:=2.7, \Rz:=0), v200, z200, Tooldata_7;
MoveJ RelTool (starting_position, 145, 270, -222 \Rx:=-2.5, \Ry:=1.8, \Rz:=0), v200, z200, Tooldata_7;
MoveJ RelTool (starting_position, 140, 269.9, -220 \Rx:=-2.4, \Ry:=0.9, \Rz:=0), v200, z200, Tooldata_7;
MoveJ RelTool (starting_position, 135, 269.9, -218 \Rx:=-2.3, \Ry:=0.3, \Rz:=0), v200, z200, Tooldata_7;
MoveJ RelTool (starting_position, 130, 269.8, -216 \Rx:=-2.2, \Ry:=-0.6, \Rz:=0), v200, z200, Tooldata_7;
MoveJ RelTool (starting_position, 125, 269.7, -214 \Rx:=-2, \Ry:=-1.5, \Rz:=0), v200, z200, Tooldata_7;
MoveJ RelTool (starting_position, 120, 269.7, -211 \Rx:=-1.8, \Ry:=-2.4, \Rz:=0), v200, z200, Tooldata_7;
MoveJ RelTool (starting_position, 115, 269.6, -209 \Rx:=-1.6, \Ry:=-3.3, \Rz:=0), v200, z200, Tooldata_7;
MoveJ RelTool (starting_position, 110, 269.5, -207 \Rx:=-1.3, \Ry:=-4.2, \Rz:=0), v200, z200, Tooldata_7;
MoveJ RelTool (starting_position, 106, 269.3, -204 \Rx:=-1, \Ry:=-5.1, \Rz:=0), v200, z200, Tooldata_7;
MoveJ RelTool (starting_position, 101, 269.2, -202 \Rx:=-0.7, \Ry:=-5.7, \Rz:=0), v200, z200, Tooldata_7;
MoveJ RelTool (starting_position, 97, 269.1, -200 \Rx:=-0.4, \Ry:=-6.3, \Rz:=0), v200, z200, Tooldata_7;
MoveJ RelTool (starting_position, 94, 268.9, -198 \Rx:=0, \Ry:=-7.2, \Rz:=0), v200, z200, Tooldata_7;
MoveJ RelTool (starting_position, 90, 268.7, -196 \Rx:=0.4, \Ry:=-7.5, \Rz:=0), v200, z200, Tooldata_7;
MoveJ RelTool (starting_position, 87, 268.5, -194 \Rx:=0.7, \Ry:=-8.1, \Rz:=0), v200, z200, Tooldata_7;
MoveJ RelTool (starting_position, 84, 268.3, -192 \Rx:=1.2, \Ry:=-8.7, \Rz:=0), v200, z200, Tooldata_7;
MoveJ RelTool (starting_position, 81, 268.1, -190 \Rx:=1.6, \Ry:=-9, \Rz:=0), v200, z200, Tooldata_7;
MoveJ RelTool (starting_position, 77, 267.8, -188 \Rx:=2, \Ry:=-9.9, \Rz:=0), v200, z200, Tooldata_7;
MoveJ RelTool (starting_position, 74, 267.5, -186 \Rx:=2.4, \Ry:=-10.5, \Rz:=0), v200, z200, Tooldata_7;
MoveJ RelTool (starting_position, 70, 267.2, -185 \Rx:=2.9, \Ry:=-11.1, \Rz:=0), v200, z200, Tooldata_7;
MoveJ RelTool (starting_position, 67, 266.8, -183 \Rx:=3.3, \Ry:=-11.7, \Rz:=0), v200, z200, Tooldata_7;
MoveJ RelTool (starting_position, 64, 266.4, -181 \Rx:=3.7, \Ry:=-12.3, \Rz:=0), v200, z200, Tooldata_7;
MoveJ RelTool (starting_position, 62, 266, -179 \Rx:=4.2, \Ry:=-12.6, \Rz:=0), v200, z200, Tooldata_7;
MoveJ RelTool (starting_position, 60, 265.6, -177 \Rx:=4.5, \Ry:=-12.9, \Rz:=0), v200, z200, Tooldata_7;
MoveJ RelTool (starting_position, 58, 265.2, -175 \Rx:=4.8, \Ry:=-13.2, \Rz:=0), v200, z200, Tooldata_7;
MoveJ RelTool (starting_position, 56, 264.7, -173 \Rx:=4.9, \Ry:=-13.5, \Rz:=0), v200, z200, Tooldata_7;
MoveJ RelTool (starting_position, 55, 264.1, -170 \Rx:=5.1, \Ry:=-13.8, \Rz:=0), v200, z200, Tooldata_7;
MoveJ RelTool (starting_position, 54, 263.6, -168 \Rx:=5.2, \Ry:=-14.1, \Rz:=0), v200, z200, Tooldata_7;
MoveJ RelTool (starting_position, 53, 263, -165 \Rx:=5.2, \Ry:=-14.1, \Rz:=0), v200, z200, Tooldata_7;
MoveJ RelTool (starting_position, 53, 262.4, -162 \Rx:=5.1, \Ry:=-14.1, \Rz:=0), v200, z200, Tooldata_7;
MoveJ RelTool (starting_position, 53, 261.8, -159 \Rx:=4.9, \Ry:=-13.8, \Rz:=0), v200, z200, Tooldata_7;
MoveJ RelTool (starting_position, 54, 261.2, -156 \Rx:=4.6, \Ry:=-14.1, \Rz:=0), v200, z200, Tooldata_7;
MoveJ RelTool (starting_position, 55, 260.5, -153 \Rx:=4.3, \Ry:=-13.8, \Rz:=0), v200, z200, Tooldata_7;
MoveJ RelTool (starting_position, 56, 259.8, -151 \Rx:=3.9, \Ry:=-13.5, \Rz:=0), v200, z200, Tooldata_7;
MoveJ RelTool (starting_position, 58, 259.1, -148 \Rx:=3.5, \Ry:=-13.2, \Rz:=0), v200, z200, Tooldata_7;
MoveJ RelTool (starting_position, 59, 258.4, -145 \Rx:=3.1, \Ry:=-12.9, \Rz:=0), v200, z200, Tooldata_7;
MoveJ RelTool (starting_position, 61, 257.6, -143 \Rx:=2.6, \Ry:=-12.6, \Rz:=0), v200, z200, Tooldata_7;
MoveJ RelTool (starting_position, 63, 256.9, -140 \Rx:=2.2, \Ry:=-12.3, \Rz:=0), v200, z200, Tooldata_7;
MoveJ RelTool (starting_position, 65, 256.2, -138 \Rx:=1.6, \Ry:=-12, \Rz:=0), v200, z200, Tooldata_7;
MoveJ RelTool (starting_position, 67, 255.4, -136 \Rx:=1.1, \Ry:=-11.7, \Rz:=0), v200, z200, Tooldata_7;
MoveJ RelTool (starting_position, 70, 254.6, -134 \Rx:=0.7, \Ry:=-11.1, \Rz:=0), v200, z200, Tooldata_7;
MoveJ RelTool (starting_position, 73, 253.9, -132 \Rx:=0.2, \Ry:=-10.5, \Rz:=0), v200, z200, Tooldata_7;
MoveJ RelTool (starting_position, 75, 253.1, -131 \Rx:=-0.1, \Ry:=-10.2, \Rz:=0), v200, z200, Tooldata_7;
MoveJ RelTool (starting_position, 78, 252.4, -129 \Rx:=-0.5, \Ry:=-9.6, \Rz:=0), v200, z200, Tooldata_7;
MoveJ RelTool (starting_position, 81, 251.7, -128 \Rx:=-0.7, \Ry:=-9, \Rz:=0), v200, z200, Tooldata_7;
MoveJ RelTool (starting_position, 84, 250.9, -127 \Rx:=-0.9, \Ry:=-8.7, \Rz:=0), v200, z200, Tooldata_7;
MoveJ RelTool (starting_position, 87, 250.2, -126 \Rx:=-1, \Ry:=-8.1, \Rz:=0), v200, z200, Tooldata_7;
MoveJ RelTool (starting_position, 90, 249.5, -125 \Rx:=-1.1, \Ry:=-7.5, \Rz:=0), v200, z200, Tooldata_7;
MoveJ RelTool (starting_position, 92, 248.9, -125 \Rx:=-1.1, \Ry:=-7.2, \Rz:=0), v200, z200, Tooldata_7;
MoveJ RelTool (starting_position, 94, 248.2, -125 \Rx:=-1, \Ry:=-6.6, \Rz:=0), v200, z200, Tooldata_7;
MoveJ RelTool (starting_position, 97, 247.6, -124 \Rx:=-0.8, \Ry:=-6.3, \Rz:=0), v200, z200, Tooldata_7;
MoveJ RelTool (starting_position, 98, 247, -124 \Rx:=-0.5, \Ry:=-6, \Rz:=0), v200, z200, Tooldata_7;
MoveJ RelTool (starting_position, 100, 246.4, -124 \Rx:=-0.2, \Ry:=-6, \Rz:=0), v200, z200, Tooldata_7;
MoveJ RelTool (starting_position, 102, 245.9, -124 \Rx:=0.1, \Ry:=-5.7, \Rz:=0), v200, z200, Tooldata_7;
MoveJ RelTool (starting_position, 104, 245.4, -124 \Rx:=0.6, \Ry:=-5.1, \Rz:=0), v200, z200, Tooldata_7;
MoveJ RelTool (starting_position, 105, 244.9, -124 \Rx:=1, \Ry:=-4.8, \Rz:=0), v200, z200, Tooldata_7;
MoveJ RelTool (starting_position, 107, 244.4, -124 \Rx:=1.5, \Ry:=-4.5, \Rz:=0), v200, z200, Tooldata_7;
MoveJ RelTool (starting_position, 108, 244, -124 \Rx:=2, \Ry:=-4.2, \Rz:=0), v200, z200, Tooldata_7;
MoveJ RelTool (starting_position, 109, 243.6, -124 \Rx:=2.5, \Ry:=-4.2, \Rz:=0), v200, z200, Tooldata_7;
MoveJ RelTool (starting_position, 110, 243.2, -124 \Rx:=2.9, \Ry:=-4.2, \Rz:=0), v200, z200, Tooldata_7;
MoveJ RelTool (starting_position, 110, 242.9, -124 \Rx:=3.3, \Ry:=-4.2, \Rz:=0), v200, z200, Tooldata_7;
MoveJ RelTool (starting_position, 111, 242.5, -124 \Rx:=3.7, \Ry:=-3.9, \Rz:=0), v200, z200, Tooldata_7;
MoveJ RelTool (starting_position, 112, 242.3, -124 \Rx:=4.1, \Ry:=-3.6, \Rz:=0), v200, z200, Tooldata_7;
MoveJ RelTool (starting_position, 113, 242, -124 \Rx:=4.5, \Ry:=-3.6, \Rz:=0), v200, z200, Tooldata_7;
MoveJ RelTool (starting_position, 113, 241.7, -124 \Rx:=4.7, \Ry:=-3.6, \Rz:=0), v200, z200, Tooldata_7;
MoveJ RelTool (starting_position, 114, 241.5, -124 \Rx:=5, \Ry:=-3.3, \Rz:=0), v200, z200, Tooldata_7;
MoveJ RelTool (starting_position, 114, 241.3, -123 \Rx:=5.1, \Ry:=-3.3, \Rz:=0), v200, z200, Tooldata_7;
MoveJ RelTool (starting_position, 115, 241.1, -123 \Rx:=5.3, \Ry:=-3.3, \Rz:=0), v200, z200, Tooldata_7;
MoveJ RelTool (starting_position, 116, 241, -123 \Rx:=5.4, \Ry:=-3.3, \Rz:=0), v200, z200, Tooldata_7;
MoveJ RelTool (starting_position, 116, 240.8, -122 \Rx:=5.4, \Ry:=-3, \Rz:=0), v200, z200, Tooldata_7;
MoveJ RelTool (starting_position, 117, 240.7, -122 \Rx:=5.4, \Ry:=-3, \Rz:=0), v200, z200, Tooldata_7;
MoveJ RelTool (starting_position, 119, 240.6, -121 \Rx:=5.5, \Ry:=-2.7, \Rz:=0), v200, z200, Tooldata_7;
MoveJ RelTool (starting_position, 120, 240.5, -121 \Rx:=5.5, \Ry:=-2.4, \Rz:=0), v200, z200, Tooldata_7;
MoveJ RelTool (starting_position, 122, 240.4, -120 \Rx:=5.6, \Ry:=-2.1, \Rz:=0), v200, z200, Tooldata_7;
MoveJ RelTool (starting_position, 123, 240.3, -119 \Rx:=5.6, \Ry:=-1.8, \Rz:=0), v200, z200, Tooldata_7;
MoveJ RelTool (starting_position, 125, 240.2, -119 \Rx:=5.5, \Ry:=-1.5, \Rz:=0), v200, z200, Tooldata_7;
MoveJ RelTool (starting_position, 127, 240.2, -118 \Rx:=5.5, \Ry:=-1.2, \Rz:=0), v200, z200, Tooldata_7;
MoveJ RelTool (starting_position, 129, 240.1, -117 \Rx:=5.6, \Ry:=-0.9, \Rz:=0), v200, z200, Tooldata_7;
MoveJ RelTool (starting_position, 131, 240.1, -117 \Rx:=5.7, \Ry:=-0.3, \Rz:=0), v200, z200, Tooldata_7;
MoveJ RelTool (starting_position, 133, 240, -116 \Rx:=5.8, \Ry:=-0, \Rz:=0), v200, z200, Tooldata_7;
MoveJ RelTool (starting_position, 135, 240, -115 \Rx:=6, \Ry:=0.3, \Rz:=0), v200, z200, Tooldata_7;
MoveJ RelTool (starting_position, 137, 240, -114 \Rx:=6.2, \Ry:=0.6, \Rz:=0), v200, z200, Tooldata_7;
MoveJ RelTool (starting_position, 139, 240, -113 \Rx:=6.3, \Ry:=0.9, \Rz:=0), v200, z200, Tooldata_7;
MoveJ RelTool (starting_position, 141, 240, -113 \Rx:=6.5, \Ry:=1.2, \Rz:=0), v200, z200, Tooldata_7;
MoveJ RelTool (starting_position, 143, 240, -112 \Rx:=6.7, \Ry:=1.5, \Rz:=0), v200, z200, Tooldata_7;
MoveJ RelTool (starting_position, 146, 240, -111 \Rx:=6.9, \Ry:=2.1, \Rz:=0), v200, z200, Tooldata_7;
MoveJ RelTool (starting_position, 149, 240, -111 \Rx:=7, \Ry:=2.7, \Rz:=0), v200, z200, Tooldata_7;
MoveJ RelTool (starting_position, 152, 240, -111 \Rx:=7.1, \Ry:=3, \Rz:=0), v200, z200, Tooldata_7;
MoveJ RelTool (starting_position, 155, 240, -110 \Rx:=7.2, \Ry:=3.6, \Rz:=0), v200, z200, Tooldata_7;
MoveJ RelTool (starting_position, 159, 240, -110 \Rx:=7.2, \Ry:=4.2, \Rz:=0), v200, z200, Tooldata_7;
MoveJ RelTool (starting_position, 162, 240, -111 \Rx:=7.2, \Ry:=5.1, \Rz:=0), v200, z200, Tooldata_7;
MoveJ RelTool (starting_position, 166, 240, -111 \Rx:=7.2, \Ry:=5.7, \Rz:=0), v200, z200, Tooldata_7;
MoveJ RelTool (starting_position, 170, 240, -112 \Rx:=7.1, \Ry:=6.3, \Rz:=0), v200, z200, Tooldata_7;
MoveJ RelTool (starting_position, 174, 240, -113 \Rx:=7, \Ry:=6.9, \Rz:=0), v200, z200, Tooldata_7;
MoveJ RelTool (starting_position, 178, 240, -114 \Rx:=6.9, \Ry:=7.5, \Rz:=0), v200, z200, Tooldata_7;
MoveJ RelTool (starting_position, 181, 240, -115 \Rx:=6.8, \Ry:=8.4, \Rz:=0), v200, z200, Tooldata_7;
MoveJ RelTool (starting_position, 185, 240, -117 \Rx:=6.6, \Ry:=9, \Rz:=0), v200, z200, Tooldata_7;
MoveJ RelTool (starting_position, 188, 240, -119 \Rx:=6.4, \Ry:=9.6, \Rz:=0), v200, z200, Tooldata_7;
MoveJ RelTool (starting_position, 192, 240, -121 \Rx:=6.2, \Ry:=10.2, \Rz:=0), v200, z200, Tooldata_7;
MoveJ RelTool (starting_position, 194, 240, -124 \Rx:=6, \Ry:=10.5, \Rz:=0), v200, z200, Tooldata_7;
MoveJ RelTool (starting_position, 197, 240, -126 \Rx:=5.8, \Ry:=11.1, \Rz:=0), v200, z200, Tooldata_7;
MoveJ RelTool (starting_position, 199, 240, -129 \Rx:=5.7, \Ry:=11.4, \Rz:=0), v200, z200, Tooldata_7;
MoveJ RelTool (starting_position, 201, 240, -132 \Rx:=5.5, \Ry:=12, \Rz:=0), v200, z200, Tooldata_7;
MoveJ RelTool (starting_position, 203, 239.9, -134 \Rx:=5.4, \Ry:=12, \Rz:=0), v200, z200, Tooldata_7;
MoveJ RelTool (starting_position, 204, 239.9, -137 \Rx:=5.3, \Ry:=12.3, \Rz:=0), v200, z200, Tooldata_7;
MoveJ RelTool (starting_position, 204, 239.8, -140 \Rx:=5.3, \Ry:=12.3, \Rz:=0), v200, z200, Tooldata_7;
MoveJ RelTool (starting_position, 205, 239.7, -143 \Rx:=5.3, \Ry:=12.3, \Rz:=0), v200, z200, Tooldata_7;
MoveJ RelTool (starting_position, 205, 239.7, -146 \Rx:=5.4, \Ry:=12.3, \Rz:=0), v200, z200, Tooldata_7;
MoveJ RelTool (starting_position, 205, 239.6, -149 \Rx:=5.5, \Ry:=12.3, \Rz:=0), v200, z200, Tooldata_7;
MoveJ RelTool (starting_position, 204, 239.5, -151 \Rx:=5.6, \Ry:=12.3, \Rz:=0), v200, z200, Tooldata_7;
MoveJ RelTool (starting_position, 204, 239.3, -154 \Rx:=5.8, \Ry:=12.3, \Rz:=0), v200, z200, Tooldata_7;
MoveJ RelTool (starting_position, 203, 239.2, -156 \Rx:=6.1, \Ry:=12, \Rz:=0), v200, z200, Tooldata_7;
MoveJ RelTool (starting_position, 202, 239.1, -158 \Rx:=6.4, \Ry:=12, \Rz:=0), v200, z200, Tooldata_7;
MoveJ RelTool (starting_position, 201, 238.9, -159 \Rx:=6.6, \Ry:=11.7, \Rz:=0), v200, z200, Tooldata_7;
MoveJ RelTool (starting_position, 200, 238.7, -161 \Rx:=6.9, \Ry:=11.4, \Rz:=0), v200, z200, Tooldata_7;
MoveJ RelTool (starting_position, 199, 238.5, -161 \Rx:=7.3, \Ry:=11.4, \Rz:=0), v200, z200, Tooldata_7;
MoveJ RelTool (starting_position, 198, 238.3, -162 \Rx:=7.6, \Ry:=11.1, \Rz:=0), v200, z200, Tooldata_7;
MoveJ RelTool (starting_position, 196, 238.1, -162 \Rx:=8, \Ry:=10.8, \Rz:=0), v200, z200, Tooldata_7;
MoveJ RelTool (starting_position, 195, 237.8, -162 \Rx:=8.3, \Ry:=10.5, \Rz:=0), v200, z200, Tooldata_7;
MoveJ RelTool (starting_position, 194, 237.5, -161 \Rx:=8.7, \Ry:=10.5, \Rz:=0), v200, z200, Tooldata_7;
MoveJ RelTool (starting_position, 193, 237.2, -160 \Rx:=9.1, \Ry:=10.2, \Rz:=0), v200, z200, Tooldata_7;
MoveJ RelTool (starting_position, 192, 236.8, -159 \Rx:=9.5, \Ry:=9.9, \Rz:=0), v200, z200, Tooldata_7;
MoveJ RelTool (starting_position, 191, 236.4, -158 \Rx:=9.9, \Ry:=9.9, \Rz:=0), v200, z200, Tooldata_7;
MoveJ RelTool (starting_position, 190, 236, -156 \Rx:=10.3, \Ry:=9.6, \Rz:=0), v200, z200, Tooldata_7;
MoveJ RelTool (starting_position, 190, 235.6, -154 \Rx:=10.6, \Ry:=9.6, \Rz:=0), v200, z200, Tooldata_7;
MoveJ RelTool (starting_position, 190, 235.2, -153 \Rx:=11, \Ry:=9.6, \Rz:=0), v200, z200, Tooldata_7;
MoveJ RelTool (starting_position, 190, 234.7, -151 \Rx:=11.3, \Ry:=9.6, \Rz:=0), v200, z200, Tooldata_7;
MoveJ RelTool (starting_position, 190, 234.1, -149 \Rx:=11.6, \Ry:=9.9, \Rz:=0), v200, z200, Tooldata_7;
MoveJ RelTool (starting_position, 190, 233.6, -148 \Rx:=11.8, \Ry:=9.6, \Rz:=0), v200, z200, Tooldata_7;
MoveJ RelTool (starting_position, 190, 233, -146 \Rx:=12, \Ry:=9.6, \Rz:=0), v200, z200, Tooldata_7;
MoveJ RelTool (starting_position, 190, 232.4, -145 \Rx:=12.2, \Ry:=9.6, \Rz:=0), v200, z200, Tooldata_7;
MoveJ RelTool (starting_position, 191, 231.8, -144 \Rx:=12.4, \Ry:=9.9, \Rz:=0), v200, z200, Tooldata_7;
MoveJ RelTool (starting_position, 192, 231.2, -144 \Rx:=12.6, \Ry:=10.2, \Rz:=0), v200, z200, Tooldata_7;
MoveJ RelTool (starting_position, 192, 230.5, -143 \Rx:=12.7, \Ry:=10.2, \Rz:=0), v200, z200, Tooldata_7;
MoveJ RelTool (starting_position, 193, 229.8, -143 \Rx:=12.8, \Ry:=10.2, \Rz:=0), v200, z200, Tooldata_7;
MoveJ RelTool (starting_position, 194, 229.1, -143 \Rx:=12.9, \Ry:=10.5, \Rz:=0), v200, z200, Tooldata_7;
MoveJ RelTool (starting_position, 195, 228.4, -143 \Rx:=13.1, \Ry:=10.5, \Rz:=0), v200, z200, Tooldata_7;
MoveJ RelTool (starting_position, 197, 227.6, -144 \Rx:=13.2, \Ry:=10.8, \Rz:=0), v200, z200, Tooldata_7;
MoveJ RelTool (starting_position, 199, 226.9, -144 \Rx:=13.4, \Ry:=11.1, \Rz:=0), v200, z200, Tooldata_7;
MoveJ RelTool (starting_position, 201, 226.2, -145 \Rx:=13.5, \Ry:=11.7, \Rz:=0), v200, z200, Tooldata_7;
MoveJ RelTool (starting_position, 203, 225.4, -146 \Rx:=13.6, \Ry:=12, \Rz:=0), v200, z200, Tooldata_7;
MoveJ RelTool (starting_position, 205, 224.6, -147 \Rx:=13.7, \Ry:=12.3, \Rz:=0), v200, z200, Tooldata_7;
MoveJ RelTool (starting_position, 206, 223.9, -148 \Rx:=13.8, \Ry:=12.6, \Rz:=0), v200, z200, Tooldata_7;
MoveJ RelTool (starting_position, 208, 223.1, -149 \Rx:=13.9, \Ry:=12.9, \Rz:=0), v200, z200, Tooldata_7;
MoveJ RelTool (starting_position, 211, 222.4, -150 \Rx:=14, \Ry:=13.2, \Rz:=0), v200, z200, Tooldata_7;
MoveJ RelTool (starting_position, 213, 221.7, -151 \Rx:=14, \Ry:=13.8, \Rz:=0), v200, z200, Tooldata_7;
MoveJ RelTool (starting_position, 215, 220.9, -153 \Rx:=14.1, \Ry:=14.1, \Rz:=0), v200, z200, Tooldata_7;
MoveJ RelTool (starting_position, 217, 220.2, -154 \Rx:=14.1, \Ry:=14.4, \Rz:=0), v200, z200, Tooldata_7;
MoveJ RelTool (starting_position, 219, 219.5, -156 \Rx:=14.2, \Ry:=15, \Rz:=0), v200, z200, Tooldata_7;
MoveJ RelTool (starting_position, 221, 218.9, -158 \Rx:=14.1, \Ry:=15.3, \Rz:=0), v200, z200, Tooldata_7;
MoveJ RelTool (starting_position, 222, 218.2, -159 \Rx:=14.1, \Ry:=15.3, \Rz:=0), v200, z200, Tooldata_7;
MoveJ RelTool (starting_position, 223, 217.6, -161 \Rx:=14, \Ry:=15.6, \Rz:=0), v200, z200, Tooldata_7;
MoveJ RelTool (starting_position, 225, 217, -163 \Rx:=14, \Ry:=15.6, \Rz:=0), v200, z200, Tooldata_7;
MoveJ RelTool (starting_position, 226, 216.4, -165 \Rx:=13.8, \Ry:=15.9, \Rz:=0), v200, z200, Tooldata_7;
MoveJ RelTool (starting_position, 227, 215.9, -167 \Rx:=13.7, \Ry:=16.2, \Rz:=0), v200, z200, Tooldata_7;
MoveJ RelTool (starting_position, 229, 215.4, -169 \Rx:=13.6, \Ry:=16.5, \Rz:=0), v200, z200, Tooldata_7;
MoveJ RelTool (starting_position, 230, 214.9, -171 \Rx:=13.4, \Ry:=16.8, \Rz:=0), v200, z200, Tooldata_7;
MoveJ RelTool (starting_position, 232, 214.4, -173 \Rx:=13.3, \Ry:=17.1, \Rz:=0), v200, z200, Tooldata_7;
MoveJ RelTool (starting_position, 233, 214, -175 \Rx:=13.1, \Ry:=17.1, \Rz:=0), v200, z200, Tooldata_7;
MoveJ RelTool (starting_position, 235, 213.6, -177 \Rx:=13, \Ry:=17.4, \Rz:=0), v200, z200, Tooldata_7;
MoveJ RelTool (starting_position, 237, 213.2, -179 \Rx:=12.9, \Ry:=18, \Rz:=0), v200, z200, Tooldata_7;
MoveJ RelTool (starting_position, 240, 212.9, -181 \Rx:=12.7, \Ry:=18.3, \Rz:=0), v200, z200, Tooldata_7;
MoveJ RelTool (starting_position, 242, 212.5, -183 \Rx:=12.6, \Ry:=18.9, \Rz:=0), v200, z200, Tooldata_7;
MoveJ RelTool (starting_position, 244, 212.3, -185 \Rx:=12.5, \Ry:=19.2, \Rz:=0), v200, z200, Tooldata_7;
MoveJ RelTool (starting_position, 245, 212, -187 \Rx:=12.5, \Ry:=19.5, \Rz:=0), v200, z200, Tooldata_7;
MoveJ RelTool (starting_position, 246, 211.7, -190 \Rx:=12.4, \Ry:=19.5, \Rz:=0), v200, z200, Tooldata_7;
MoveJ RelTool (starting_position, 247, 211.5, -192 \Rx:=12.4, \Ry:=19.5, \Rz:=0), v200, z200, Tooldata_7;
MoveJ RelTool (starting_position, 247, 211.3, -194 \Rx:=12.4, \Ry:=19.8, \Rz:=0), v200, z200, Tooldata_7;
MoveJ RelTool (starting_position, 248, 211.1, -196 \Rx:=12.3, \Ry:=19.8, \Rz:=0), v200, z200, Tooldata_7;
MoveJ RelTool (starting_position, 248, 211, -199 \Rx:=12.3, \Ry:=19.8, \Rz:=0), v200, z200, Tooldata_7;
MoveJ RelTool (starting_position, 248, 210.8, -201 \Rx:=12.3, \Ry:=19.8, \Rz:=0), v200, z200, Tooldata_7;
MoveJ RelTool (starting_position, 248, 210.7, -203 \Rx:=12.4, \Ry:=19.8, \Rz:=0), v200, z200, Tooldata_7;
MoveJ RelTool (starting_position, 249, 210.6, -206 \Rx:=12.4, \Ry:=19.8, \Rz:=0), v200, z200, Tooldata_7;
MoveJ RelTool (starting_position, 249, 210.5, -208 \Rx:=12.5, \Ry:=20.1, \Rz:=0), v200, z200, Tooldata_7;
MoveJ RelTool (starting_position, 249, 210.4, -211 \Rx:=12.5, \Ry:=20.1, \Rz:=0), v200, z200, Tooldata_7;
MoveJ RelTool (starting_position, 250, 210.3, -213 \Rx:=12.6, \Ry:=20.1, \Rz:=0), v200, z200, Tooldata_7;
MoveJ RelTool (starting_position, 250, 210.2, -215 \Rx:=12.6, \Ry:=20.1, \Rz:=0), v200, z200, Tooldata_7;
MoveJ RelTool (starting_position, 250, 210.2, -218 \Rx:=12.7, \Ry:=20.1, \Rz:=0), v200, z200, Tooldata_7;
MoveJ RelTool (starting_position, 251, 210.1, -221 \Rx:=12.8, \Ry:=20.4, \Rz:=0), v200, z200, Tooldata_7;
MoveJ RelTool (starting_position, 251, 210.1, -223 \Rx:=12.8, \Ry:=20.4, \Rz:=0), v200, z200, Tooldata_7;
MoveJ RelTool (starting_position, 251, 210, -226 \Rx:=12.9, \Ry:=20.4, \Rz:=0), v200, z200, Tooldata_7;
MoveJ RelTool (starting_position, 252, 210, -228 \Rx:=12.9, \Ry:=20.4, \Rz:=0), v200, z200, Tooldata_7;
MoveJ RelTool (starting_position, 252, 210, -231 \Rx:=12.9, \Ry:=20.4, \Rz:=0), v200, z200, Tooldata_7;
MoveJ RelTool (starting_position, 252, 210, -234 \Rx:=13, \Ry:=20.7, \Rz:=0), v200, z200, Tooldata_7;
MoveJ RelTool (starting_position, 252, 210, -237 \Rx:=13, \Ry:=20.7, \Rz:=0), v200, z200, Tooldata_7;
MoveJ RelTool (starting_position, 252, 210, -240 \Rx:=13, \Ry:=20.7, \Rz:=0), v200, z200, Tooldata_7;
MoveJ RelTool (starting_position, 252, 210, -242 \Rx:=13, \Ry:=20.4, \Rz:=0), v200, z200, Tooldata_7;
MoveJ RelTool (starting_position, 252, 209.9, -245 \Rx:=12.9, \Ry:=20.4, \Rz:=0), v200, z200, Tooldata_7;
MoveJ RelTool (starting_position, 251, 209.9, -249 \Rx:=12.8, \Ry:=20.4, \Rz:=0), v200, z200, Tooldata_7;
MoveJ RelTool (starting_position, 251, 209.8, -252 \Rx:=12.7, \Ry:=20.4, \Rz:=0), v200, z200, Tooldata_7;
MoveJ RelTool (starting_position, 250, 209.7, -255 \Rx:=12.5, \Ry:=20.1, \Rz:=0), v200, z200, Tooldata_7;
MoveJ RelTool (starting_position, 249, 209.7, -258 \Rx:=12.3, \Ry:=20.1, \Rz:=0), v200, z200, Tooldata_7;
MoveJ RelTool (starting_position, 248, 209.6, -262 \Rx:=12.1, \Ry:=19.8, \Rz:=0), v200, z200, Tooldata_7;
MoveJ RelTool (starting_position, 247, 209.5, -265 \Rx:=11.9, \Ry:=19.8, \Rz:=0), v200, z200, Tooldata_7;
MoveJ RelTool (starting_position, 246, 209.3, -269 \Rx:=11.7, \Ry:=19.5, \Rz:=0), v200, z200, Tooldata_7;
MoveJ RelTool (starting_position, 245, 209.2, -272 \Rx:=11.4, \Ry:=19.2, \Rz:=0), v200, z200, Tooldata_7;
MoveJ RelTool (starting_position, 244, 209.1, -276 \Rx:=11.1, \Ry:=19.2, \Rz:=0), v200, z200, Tooldata_7;
MoveJ RelTool (starting_position, 243, 208.9, -279 \Rx:=10.8, \Ry:=18.9, \Rz:=0), v200, z200, Tooldata_7;
MoveJ RelTool (starting_position, 242, 208.7, -283 \Rx:=10.4, \Ry:=18.6, \Rz:=0), v200, z200, Tooldata_7;
MoveJ RelTool (starting_position, 241, 208.5, -287 \Rx:=10.1, \Ry:=18.6, \Rz:=0), v200, z200, Tooldata_7;
MoveJ RelTool (starting_position, 240, 208.3, -290 \Rx:=9.7, \Ry:=18.3, \Rz:=0), v200, z200, Tooldata_7;
MoveJ RelTool (starting_position, 239, 208.1, -293 \Rx:=9.2, \Ry:=18.3, \Rz:=0), v200, z200, Tooldata_7;
MoveJ RelTool (starting_position, 238, 207.8, -297 \Rx:=8.7, \Ry:=18, \Rz:=0), v200, z200, Tooldata_7;
MoveJ RelTool (starting_position, 237, 207.5, -300 \Rx:=8.2, \Ry:=17.7, \Rz:=0), v200, z200, Tooldata_7;
MoveJ RelTool (starting_position, 236, 207.2, -303 \Rx:=7.8, \Ry:=17.7, \Rz:=0), v200, z200, Tooldata_7;
MoveJ RelTool (starting_position, 235, 206.8, -305 \Rx:=7.3, \Ry:=17.4, \Rz:=0), v200, z200, Tooldata_7;
MoveJ RelTool (starting_position, 234, 206.4, -308 \Rx:=6.8, \Ry:=17.4, \Rz:=0), v200, z200, Tooldata_7;
MoveJ RelTool (starting_position, 233, 206, -310 \Rx:=6.3, \Ry:=17.1, \Rz:=0), v200, z200, Tooldata_7;
MoveJ RelTool (starting_position, 232, 205.6, -313 \Rx:=5.9, \Ry:=16.8, \Rz:=0), v200, z200, Tooldata_7;
MoveJ RelTool (starting_position, 231, 205.2, -315 \Rx:=5.4, \Ry:=16.8, \Rz:=0), v200, z200, Tooldata_7;
MoveJ RelTool (starting_position, 230, 204.7, -316 \Rx:=5, \Ry:=16.8, \Rz:=0), v200, z200, Tooldata_7;
MoveJ RelTool (starting_position, 230, 204.1, -318 \Rx:=4.6, \Ry:=16.5, \Rz:=0), v200, z200, Tooldata_7;
MoveJ RelTool (starting_position, 230, 203.6, -320 \Rx:=4.3, \Ry:=16.5, \Rz:=0), v200, z200, Tooldata_7;
MoveJ RelTool (starting_position, 230, 203, -321 \Rx:=4.1, \Ry:=16.5, \Rz:=0), v200, z200, Tooldata_7;
MoveJ RelTool (starting_position, 230, 202.4, -323 \Rx:=3.9, \Ry:=16.8, \Rz:=0), v200, z200, Tooldata_7;
MoveJ RelTool (starting_position, 230, 201.8, -324 \Rx:=3.8, \Ry:=16.8, \Rz:=0), v200, z200, Tooldata_7;
MoveJ RelTool (starting_position, 231, 201.2, -325 \Rx:=3.8, \Ry:=16.8, \Rz:=0), v200, z200, Tooldata_7;
MoveJ RelTool (starting_position, 231, 200.5, -326 \Rx:=3.8, \Ry:=16.8, \Rz:=0), v200, z200, Tooldata_7;
MoveJ RelTool (starting_position, 232, 199.8, -328 \Rx:=3.9, \Ry:=16.8, \Rz:=0), v200, z200, Tooldata_7;
MoveJ RelTool (starting_position, 232, 199.1, -329 \Rx:=4.1, \Ry:=17.1, \Rz:=0), v200, z200, Tooldata_7;
MoveJ RelTool (starting_position, 233, 198.4, -330 \Rx:=4.4, \Ry:=17.1, \Rz:=0), v200, z200, Tooldata_7;
MoveJ RelTool (starting_position, 235, 197.6, -331 \Rx:=4.7, \Ry:=17.4, \Rz:=0), v200, z200, Tooldata_7;
MoveJ RelTool (starting_position, 236, 196.9, -333 \Rx:=5.1, \Ry:=17.7, \Rz:=0), v200, z200, Tooldata_7;
MoveJ RelTool (starting_position, 238, 196.2, -334 \Rx:=5.6, \Ry:=18, \Rz:=0), v200, z200, Tooldata_7;
MoveJ RelTool (starting_position, 240, 195.4, -336 \Rx:=6.1, \Ry:=18.3, \Rz:=0), v200, z200, Tooldata_7;
MoveJ RelTool (starting_position, 242, 194.6, -338 \Rx:=6.7, \Ry:=18.9, \Rz:=0), v200, z200, Tooldata_7;
MoveJ RelTool (starting_position, 244, 193.9, -339 \Rx:=7.3, \Ry:=19.2, \Rz:=0), v200, z200, Tooldata_7;
MoveJ RelTool (starting_position, 246, 193.1, -341 \Rx:=7.9, \Ry:=19.5, \Rz:=0), v200, z200, Tooldata_7;
MoveJ RelTool (starting_position, 248, 192.4, -343 \Rx:=8.4, \Ry:=19.8, \Rz:=0), v200, z200, Tooldata_7;
MoveJ RelTool (starting_position, 250, 191.7, -346 \Rx:=9, \Ry:=20.1, \Rz:=0), v200, z200, Tooldata_7;
MoveJ RelTool (starting_position, 251, 190.9, -348 \Rx:=9.5, \Ry:=20.4, \Rz:=0), v200, z200, Tooldata_7;
MoveJ RelTool (starting_position, 253, 190.2, -351 \Rx:=10, \Ry:=20.7, \Rz:=0), v200, z200, Tooldata_7;
MoveJ RelTool (starting_position, 254, 189.5, -354 \Rx:=10.5, \Ry:=21, \Rz:=0), v200, z200, Tooldata_7;
MoveJ RelTool (starting_position, 255, 188.9, -357 \Rx:=10.9, \Ry:=21.3, \Rz:=0), v200, z200, Tooldata_7;
MoveJ RelTool (starting_position, 256, 188.2, -360 \Rx:=11.2, \Ry:=21.3, \Rz:=0), v200, z200, Tooldata_7;
MoveJ RelTool (starting_position, 256, 187.6, -364 \Rx:=11.4, \Ry:=21.3, \Rz:=0), v200, z200, Tooldata_7;
MoveJ RelTool (starting_position, 257, 187, -367 \Rx:=11.6, \Ry:=21.3, \Rz:=0), v200, z200, Tooldata_7;
MoveJ RelTool (starting_position, 257, 186.4, -371 \Rx:=11.7, \Ry:=21.3, \Rz:=0), v200, z200, Tooldata_7;
MoveJ RelTool (starting_position, 256, 185.9, -374 \Rx:=11.7, \Ry:=21.3, \Rz:=0), v200, z200, Tooldata_7;
MoveJ RelTool (starting_position, 256, 185.4, -378 \Rx:=11.7, \Ry:=21.3, \Rz:=0), v200, z200, Tooldata_7;
MoveJ RelTool (starting_position, 255, 184.9, -381 \Rx:=11.5, \Ry:=21, \Rz:=0), v200, z200, Tooldata_7;
MoveJ RelTool (starting_position, 254, 184.4, -385 \Rx:=11.3, \Ry:=21, \Rz:=0), v200, z200, Tooldata_7;
MoveJ RelTool (starting_position, 252, 184, -388 \Rx:=11, \Ry:=20.7, \Rz:=0), v200, z200, Tooldata_7;
MoveJ RelTool (starting_position, 251, 183.6, -392 \Rx:=10.6, \Ry:=20.4, \Rz:=0), v200, z200, Tooldata_7;
MoveJ RelTool (starting_position, 249, 183.2, -395 \Rx:=10.2, \Ry:=19.8, \Rz:=0), v200, z200, Tooldata_7;
MoveJ RelTool (starting_position, 246, 182.9, -399 \Rx:=9.7, \Ry:=19.5, \Rz:=0), v200, z200, Tooldata_7;
MoveJ RelTool (starting_position, 244, 182.5, -402 \Rx:=9.2, \Ry:=19.2, \Rz:=0), v200, z200, Tooldata_7;
MoveJ RelTool (starting_position, 241, 182.3, -405 \Rx:=8.7, \Ry:=18.6, \Rz:=0), v200, z200, Tooldata_7;
MoveJ RelTool (starting_position, 239, 182, -407 \Rx:=8.1, \Ry:=18.3, \Rz:=0), v200, z200, Tooldata_7;
MoveJ RelTool (starting_position, 235, 181.7, -410 \Rx:=7.5, \Ry:=17.7, \Rz:=0), v200, z200, Tooldata_7;
MoveJ RelTool (starting_position, 232, 181.5, -412 \Rx:=6.9, \Ry:=17.1, \Rz:=0), v200, z200, Tooldata_7;
MoveJ RelTool (starting_position, 228, 181.3, -414 \Rx:=6.4, \Ry:=16.5, \Rz:=0), v200, z200, Tooldata_7;
MoveJ RelTool (starting_position, 225, 181.1, -416 \Rx:=5.8, \Ry:=15.6, \Rz:=0), v200, z200, Tooldata_7;
MoveJ RelTool (starting_position, 221, 181, -418 \Rx:=5.3, \Ry:=15, \Rz:=0), v200, z200, Tooldata_7;
MoveJ RelTool (starting_position, 217, 180.8, -420 \Rx:=4.7, \Ry:=14.4, \Rz:=0), v200, z200, Tooldata_7;
MoveJ RelTool (starting_position, 213, 180.7, -421 \Rx:=4.3, \Ry:=13.8, \Rz:=0), v200, z200, Tooldata_7;
MoveJ RelTool (starting_position, 209, 180.6, -423 \Rx:=3.8, \Ry:=12.9, \Rz:=0), v200, z200, Tooldata_7;
MoveJ RelTool (starting_position, 205, 180.5, -424 \Rx:=3.4, \Ry:=12.3, \Rz:=0), v200, z200, Tooldata_7;
MoveJ RelTool (starting_position, 202, 180.4, -425 \Rx:=3, \Ry:=11.7, \Rz:=0), v200, z200, Tooldata_7;
MoveJ RelTool (starting_position, 198, 180.3, -426 \Rx:=2.7, \Ry:=11.1, \Rz:=0), v200, z200, Tooldata_7;
MoveJ RelTool (starting_position, 195, 180.2, -427 \Rx:=2.4, \Ry:=10.5, \Rz:=0), v200, z200, Tooldata_7;
MoveJ RelTool (starting_position, 191, 180.2, -427 \Rx:=2.1, \Ry:=9.9, \Rz:=0), v200, z200, Tooldata_7;
MoveJ RelTool (starting_position, 188, 180.1, -428 \Rx:=1.9, \Ry:=9.3, \Rz:=0), v200, z200, Tooldata_7;
MoveJ RelTool (starting_position, 185, 180, -428 \Rx:=1.7, \Ry:=8.7, \Rz:=0), v200, z200, Tooldata_7;
MoveJ RelTool (starting_position, 181, 179.9, -429 \Rx:=1.5, \Ry:=8.1, \Rz:=0), v200, z200, Tooldata_7;
MoveJ RelTool (starting_position, 179, 179.8, -429 \Rx:=1.4, \Ry:=7.8, \Rz:=0), v200, z200, Tooldata_7;
MoveJ RelTool (starting_position, 176, 179.7, -430 \Rx:=1.2, \Ry:=7.2, \Rz:=0), v200, z200, Tooldata_7;
MoveJ RelTool (starting_position, 173, 179.7, -430 \Rx:=1.1, \Ry:=6.9, \Rz:=0), v200, z200, Tooldata_7;
MoveJ RelTool (starting_position, 171, 179.6, -430 \Rx:=1.1, \Ry:=6.3, \Rz:=0), v200, z200, Tooldata_7;
MoveJ RelTool (starting_position, 169, 179.5, -431 \Rx:=1, \Ry:=6, \Rz:=0), v200, z200, Tooldata_7;
MoveJ RelTool (starting_position, 166, 179.3, -431 \Rx:=0.9, \Ry:=5.7, \Rz:=0), v200, z200, Tooldata_7;
MoveJ RelTool (starting_position, 164, 179.2, -431 \Rx:=0.9, \Ry:=5.1, \Rz:=0), v200, z200, Tooldata_7;
MoveJ RelTool (starting_position, 162, 179.1, -432 \Rx:=0.8, \Ry:=4.8, \Rz:=0), v200, z200, Tooldata_7;
MoveJ RelTool (starting_position, 160, 178.9, -432 \Rx:=0.8, \Ry:=4.5, \Rz:=0), v200, z200, Tooldata_7;
MoveJ RelTool (starting_position, 159, 178.7, -432 \Rx:=0.7, \Ry:=4.5, \Rz:=0), v200, z200, Tooldata_7;
MoveJ RelTool (starting_position, 157, 178.5, -433 \Rx:=0.6, \Ry:=3.9, \Rz:=0), v200, z200, Tooldata_7;
MoveJ RelTool (starting_position, 156, 178.3, -433 \Rx:=0.6, \Ry:=3.9, \Rz:=0), v200, z200, Tooldata_7;
MoveJ RelTool (starting_position, 154, 178.1, -433 \Rx:=0.5, \Ry:=3.6, \Rz:=0), v200, z200, Tooldata_7;
MoveJ RelTool (starting_position, 153, 177.8, -434 \Rx:=0.5, \Ry:=3.3, \Rz:=0), v200, z200, Tooldata_7;
MoveJ RelTool (starting_position, 152, 177.5, -434 \Rx:=0.5, \Ry:=3, \Rz:=0), v200, z200, Tooldata_7;
MoveJ RelTool (starting_position, 150, 177.2, -434 \Rx:=0.4, \Ry:=2.7, \Rz:=0), v200, z200, Tooldata_7;
MoveJ RelTool (starting_position, 149, 176.8, -435 \Rx:=0.4, \Ry:=2.7, \Rz:=0), v200, z200, Tooldata_7;
MoveJ RelTool (starting_position, 148, 176.4, -435 \Rx:=0.3, \Ry:=2.4, \Rz:=0), v200, z200, Tooldata_7;
MoveJ RelTool (starting_position, 147, 176, -435 \Rx:=0.3, \Ry:=2.4, \Rz:=0), v200, z200, Tooldata_7;
MoveJ RelTool (starting_position, 146, 175.6, -435 \Rx:=0.2, \Ry:=2.1, \Rz:=0), v200, z200, Tooldata_7;
MoveJ RelTool (starting_position, 146, 175.2, -436 \Rx:=0.2, \Ry:=2.1, \Rz:=0), v200, z200, Tooldata_7;
MoveJ RelTool (starting_position, 145, 174.7, -436 \Rx:=0.2, \Ry:=1.8, \Rz:=0), v200, z200, Tooldata_7;
MoveJ RelTool (starting_position, 145, 174.1, -436 \Rx:=0.2, \Ry:=1.8, \Rz:=0), v200, z200, Tooldata_7;
MoveJ RelTool (starting_position, 144, 173.6, -436 \Rx:=0.1, \Ry:=1.8, \Rz:=0), v200, z200, Tooldata_7;
MoveJ RelTool (starting_position, 144, 173, -436 \Rx:=0.1, \Ry:=1.8, \Rz:=0), v200, z200, Tooldata_7;
MoveJ RelTool (starting_position, 143, 172.4, -437 \Rx:=0.1, \Ry:=1.8, \Rz:=0), v200, z200, Tooldata_7;
MoveJ RelTool (starting_position, 143, 171.8, -437 \Rx:=0.1, \Ry:=1.5, \Rz:=0), v200, z200, Tooldata_7;
MoveJ RelTool (starting_position, 143, 171.2, -437 \Rx:=0.1, \Ry:=1.5, \Rz:=0), v200, z200, Tooldata_7;
MoveJ RelTool (starting_position, 142, 170.5, -437 \Rx:=0, \Ry:=1.5, \Rz:=0), v200, z200, Tooldata_7;
MoveJ RelTool (starting_position, 142, 169.8, -437 \Rx:=0, \Ry:=1.5, \Rz:=0), v200, z200, Tooldata_7;
MoveJ RelTool (starting_position, 142, 169.1, -437 \Rx:=0, \Ry:=1.5, \Rz:=0), v200, z200, Tooldata_7;
MoveJ RelTool (starting_position, 141, 168.4, -437 \Rx:=0, \Ry:=1.2, \Rz:=0), v200, z200, Tooldata_7;
MoveJ RelTool (starting_position, 141, 167.6, -437 \Rx:=0, \Ry:=1.2, \Rz:=0), v200, z200, Tooldata_7;
MoveJ RelTool (starting_position, 141, 166.9, -437 \Rx:=0, \Ry:=1.2, \Rz:=0), v200, z200, Tooldata_7;
MoveJ RelTool (starting_position, 141, 166.2, -437 \Rx:=0, \Ry:=1.2, \Rz:=0), v200, z200, Tooldata_7;
MoveJ RelTool (starting_position, 141, 165.4, -437 \Rx:=0, \Ry:=1.2, \Rz:=0), v200, z200, Tooldata_7;
MoveJ RelTool (starting_position, 141, 164.6, -437 \Rx:=0, \Ry:=1.2, \Rz:=0), v200, z200, Tooldata_7;
MoveJ RelTool (starting_position, 141, 163.9, -437 \Rx:=0, \Ry:=1.2, \Rz:=0), v200, z200, Tooldata_7;
MoveJ RelTool (starting_position, 141, 163.1, -437 \Rx:=0, \Ry:=1.2, \Rz:=0), v200, z200, Tooldata_7;
MoveJ RelTool (starting_position, 141, 162.4, -437 \Rx:=0, \Ry:=1.2, \Rz:=0), v200, z200, Tooldata_7;
MoveJ RelTool (starting_position, 141, 161.7, -437 \Rx:=0.1, \Ry:=1.2, \Rz:=0), v200, z200, Tooldata_7;
MoveJ RelTool (starting_position, 141, 160.9, -437 \Rx:=0.1, \Ry:=1.2, \Rz:=0), v200, z200, Tooldata_7;
MoveJ RelTool (starting_position, 142, 160.2, -437 \Rx:=0.1, \Ry:=1.5, \Rz:=0), v200, z200, Tooldata_7;
MoveJ RelTool (starting_position, 142, 159.5, -437 \Rx:=0.1, \Ry:=1.5, \Rz:=0), v200, z200, Tooldata_7;
MoveJ RelTool (starting_position, 142, 158.9, -438 \Rx:=0.1, \Ry:=1.5, \Rz:=0), v200, z200, Tooldata_7;
MoveJ RelTool (starting_position, 143, 158.2, -438 \Rx:=0.2, \Ry:=1.5, \Rz:=0), v200, z200, Tooldata_7;
MoveJ RelTool (starting_position, 143, 157.6, -438 \Rx:=0.2, \Ry:=1.5, \Rz:=0), v200, z200, Tooldata_7;
MoveJ RelTool (starting_position, 143, 157, -438 \Rx:=0.2, \Ry:=1.8, \Rz:=0), v200, z200, Tooldata_7;
MoveJ RelTool (starting_position, 144, 156.4, -438 \Rx:=0.2, \Ry:=1.8, \Rz:=0), v200, z200, Tooldata_7;
MoveJ RelTool (starting_position, 144, 155.9, -438 \Rx:=0.3, \Ry:=1.8, \Rz:=0), v200, z200, Tooldata_7;
MoveJ RelTool (starting_position, 144, 155.4, -438 \Rx:=0.3, \Ry:=1.8, \Rz:=0), v200, z200, Tooldata_7;
MoveJ RelTool (starting_position, 145, 154.9, -438 \Rx:=0.4, \Ry:=1.8, \Rz:=0), v200, z200, Tooldata_7;
MoveJ RelTool (starting_position, 145, 154.4, -438 \Rx:=0.4, \Ry:=2.1, \Rz:=0), v200, z200, Tooldata_7;
MoveJ RelTool (starting_position, 146, 154, -439 \Rx:=0.5, \Ry:=2.1, \Rz:=0), v200, z200, Tooldata_7;
MoveJ RelTool (starting_position, 146, 153.6, -439 \Rx:=0.5, \Ry:=2.1, \Rz:=0), v200, z200, Tooldata_7;
MoveJ RelTool (starting_position, 146, 153.2, -439 \Rx:=0.6, \Ry:=2.1, \Rz:=0), v200, z200, Tooldata_7;
MoveJ RelTool (starting_position, 147, 152.9, -439 \Rx:=0.6, \Ry:=2.1, \Rz:=0), v200, z200, Tooldata_7;
MoveJ RelTool (starting_position, 147, 152.5, -440 \Rx:=0.6, \Ry:=2.4, \Rz:=0), v200, z200, Tooldata_7;
MoveJ RelTool (starting_position, 147, 152.3, -440 \Rx:=0.7, \Ry:=2.4, \Rz:=0), v200, z200, Tooldata_7;
MoveJ RelTool (starting_position, 147, 152, -440 \Rx:=0.7, \Ry:=2.4, \Rz:=0), v200, z200, Tooldata_7;
MoveJ RelTool (starting_position, 148, 151.7, -441 \Rx:=0.7, \Ry:=2.4, \Rz:=0), v200, z200, Tooldata_7;
MoveJ RelTool (starting_position, 148, 151.5, -441 \Rx:=0.8, \Ry:=2.4, \Rz:=0), v200, z200, Tooldata_7;
MoveJ RelTool (starting_position, 148, 151.3, -442 \Rx:=0.8, \Ry:=2.4, \Rz:=0), v200, z200, Tooldata_7;
MoveJ RelTool (starting_position, 148, 151.1, -442 \Rx:=0.8, \Ry:=2.4, \Rz:=0), v200, z200, Tooldata_7;
MoveJ RelTool (starting_position, 148, 151, -442 \Rx:=0.8, \Ry:=2.4, \Rz:=0), v200, z200, Tooldata_7;
MoveJ RelTool (starting_position, 148, 150.8, -443 \Rx:=0.8, \Ry:=2.4, \Rz:=0), v200, z200, Tooldata_7;
MoveJ RelTool (starting_position, 148, 150.6, -443 \Rx:=0.7, \Ry:=2.4, \Rz:=0), v200, z200, Tooldata_7;
MoveJ RelTool (starting_position, 148, 150.5, -444 \Rx:=0.7, \Ry:=2.4, \Rz:=0), v200, z200, Tooldata_7;
MoveJ RelTool (starting_position, 147, 150.3, -444 \Rx:=0.7, \Ry:=2.4, \Rz:=0), v200, z200, Tooldata_7;
MoveJ RelTool (starting_position, 147, 150.2, -444 \Rx:=0.6, \Ry:=2.4, \Rz:=0), v200, z200, Tooldata_7;
MoveJ RelTool (starting_position, 147, 150, -445 \Rx:=0.6, \Ry:=2.4, \Rz:=0), v200, z200, Tooldata_7;
MoveJ RelTool (starting_position, 147, 149.9, -445 \Rx:=0.6, \Ry:=2.1, \Rz:=0), v200, z200, Tooldata_7;
MoveJ RelTool (starting_position, 146, 149.7, -445 \Rx:=0.5, \Ry:=2.1, \Rz:=0), v200, z200, Tooldata_7;
MoveJ RelTool (starting_position, 146, 149.6, -446 \Rx:=0.5, \Ry:=2.1, \Rz:=0), v200, z200, Tooldata_7;
MoveJ RelTool (starting_position, 145, 149.4, -446 \Rx:=0.4, \Ry:=2.1, \Rz:=0), v200, z200, Tooldata_7;
MoveJ RelTool (starting_position, 145, 149.2, -446 \Rx:=0.4, \Ry:=1.8, \Rz:=0), v200, z200, Tooldata_7;
MoveJ RelTool (starting_position, 144, 149.1, -446 \Rx:=0.3, \Ry:=1.8, \Rz:=0), v200, z200, Tooldata_7;
MoveJ RelTool (starting_position, 144, 148.9, -446 \Rx:=0.3, \Ry:=1.8, \Rz:=0), v200, z200, Tooldata_7;
MoveJ RelTool (starting_position, 143, 148.7, -447 \Rx:=0.2, \Ry:=1.8, \Rz:=0), v200, z200, Tooldata_7;
MoveJ RelTool (starting_position, 143, 148.5, -447 \Rx:=0.2, \Ry:=1.5, \Rz:=0), v200, z200, Tooldata_7;
MoveJ RelTool (starting_position, 142, 148.3, -447 \Rx:=0.2, \Ry:=1.5, \Rz:=0), v200, z200, Tooldata_7;
MoveJ RelTool (starting_position, 141, 148.1, -447 \Rx:=0.2, \Ry:=1.2, \Rz:=0), v200, z200, Tooldata_7;
MoveJ RelTool (starting_position, 140, 147.8, -447 \Rx:=0.1, \Ry:=1.2, \Rz:=0), v200, z200, Tooldata_7;
MoveJ RelTool (starting_position, 140, 147.5, -447 \Rx:=0.1, \Ry:=0.9, \Rz:=0), v200, z200, Tooldata_7;
MoveJ RelTool (starting_position, 139, 147.2, -447 \Rx:=0.1, \Ry:=0.9, \Rz:=0), v200, z200, Tooldata_7;
MoveJ RelTool (starting_position, 138, 146.8, -447 \Rx:=0.1, \Ry:=0.9, \Rz:=0), v200, z200, Tooldata_7;
MoveJ RelTool (starting_position, 138, 146.4, -447 \Rx:=0.1, \Ry:=0.6, \Rz:=0), v200, z200, Tooldata_7;
MoveJ RelTool (starting_position, 137, 146, -447 \Rx:=0, \Ry:=0.6, \Rz:=0), v200, z200, Tooldata_7;
MoveJ RelTool (starting_position, 136, 145.6, -447 \Rx:=0, \Ry:=0.3, \Rz:=0), v200, z200, Tooldata_7;
MoveJ RelTool (starting_position, 136, 145.2, -447 \Rx:=0, \Ry:=0.3, \Rz:=0), v200, z200, Tooldata_7;
MoveJ RelTool (starting_position, 135, 144.7, -447 \Rx:=0, \Ry:=0.3, \Rz:=0), v200, z200, Tooldata_7;
MoveJ RelTool (starting_position, 134, 144.1, -447 \Rx:=0, \Ry:=0, \Rz:=0), v200, z200, Tooldata_7;
MoveJ RelTool (starting_position, 133, 143.6, -447 \Rx:=0, \Ry:=-0, \Rz:=0), v200, z200, Tooldata_7;
MoveJ RelTool (starting_position, 133, 143, -447 \Rx:=0, \Ry:=-0.3, \Rz:=0), v200, z200, Tooldata_7;
MoveJ RelTool (starting_position, 132, 142.4, -447 \Rx:=0, \Ry:=-0.3, \Rz:=0), v200, z200, Tooldata_7;
MoveJ RelTool (starting_position, 131, 141.8, -447 \Rx:=0.1, \Ry:=-0.3, \Rz:=0), v200, z200, Tooldata_7;
MoveJ RelTool (starting_position, 131, 141.2, -447 \Rx:=0.1, \Ry:=-0.6, \Rz:=0), v200, z200, Tooldata_7;
MoveJ RelTool (starting_position, 130, 140.5, -447 \Rx:=0.2, \Ry:=-0.6, \Rz:=0), v200, z200, Tooldata_7;
MoveJ RelTool (starting_position, 129, 139.8, -447 \Rx:=0.2, \Ry:=-0.9, \Rz:=0), v200, z200, Tooldata_7;
MoveJ RelTool (starting_position, 129, 139.1, -447 \Rx:=0.2, \Ry:=-0.9, \Rz:=0), v200, z200, Tooldata_7;
MoveJ RelTool (starting_position, 128, 138.4, -447 \Rx:=0.3, \Ry:=-0.9, \Rz:=0), v200, z200, Tooldata_7;
MoveJ RelTool (starting_position, 127, 137.6, -447 \Rx:=0.3, \Ry:=-1.2, \Rz:=0), v200, z200, Tooldata_7;
MoveJ RelTool (starting_position, 126, 136.9, -447 \Rx:=0.4, \Ry:=-1.2, \Rz:=0), v200, z200, Tooldata_7;
MoveJ RelTool (starting_position, 126, 136.2, -447 \Rx:=0.5, \Ry:=-1.5, \Rz:=0), v200, z200, Tooldata_7;
MoveJ RelTool (starting_position, 125, 135.4, -447 \Rx:=0.5, \Ry:=-1.5, \Rz:=0), v200, z200, Tooldata_7;
MoveJ RelTool (starting_position, 124, 134.6, -447 \Rx:=0.6, \Ry:=-1.8, \Rz:=0), v200, z200, Tooldata_7;
MoveJ RelTool (starting_position, 124, 133.9, -447 \Rx:=0.7, \Ry:=-1.8, \Rz:=0), v200, z200, Tooldata_7;
MoveJ RelTool (starting_position, 123, 133.1, -446 \Rx:=0.8, \Ry:=-1.8, \Rz:=0), v200, z200, Tooldata_7;
MoveJ RelTool (starting_position, 123, 132.4, -446 \Rx:=0.9, \Ry:=-1.8, \Rz:=0), v200, z200, Tooldata_7;
MoveJ RelTool (starting_position, 123, 131.7, -446 \Rx:=1, \Ry:=-1.8, \Rz:=0), v200, z200, Tooldata_7;
MoveJ RelTool (starting_position, 123, 130.9, -446 \Rx:=1.1, \Ry:=-1.8, \Rz:=0), v200, z200, Tooldata_7;
MoveJ RelTool (starting_position, 122, 130.2, -446 \Rx:=1.2, \Ry:=-2.1, \Rz:=0), v200, z200, Tooldata_7;
MoveJ RelTool (starting_position, 122, 129.5, -445 \Rx:=1.2, \Ry:=-2.1, \Rz:=0), v200, z200, Tooldata_7;
MoveJ RelTool (starting_position, 122, 128.9, -445 \Rx:=1.3, \Ry:=-2.1, \Rz:=0), v200, z200, Tooldata_7;
MoveJ RelTool (starting_position, 122, 128.2, -445 \Rx:=1.4, \Ry:=-2.1, \Rz:=0), v200, z200, Tooldata_7;
MoveJ RelTool (starting_position, 122, 127.6, -444 \Rx:=1.4, \Ry:=-2.1, \Rz:=0), v200, z200, Tooldata_7;
MoveJ RelTool (starting_position, 122, 127, -444 \Rx:=1.5, \Ry:=-2.1, \Rz:=0), v200, z200, Tooldata_7;
MoveJ RelTool (starting_position, 122, 126.4, -444 \Rx:=1.6, \Ry:=-2.1, \Rz:=0), v200, z200, Tooldata_7;
MoveJ RelTool (starting_position, 122, 125.9, -443 \Rx:=1.7, \Ry:=-2.1, \Rz:=0), v200, z200, Tooldata_7;
MoveJ RelTool (starting_position, 122, 125.4, -443 \Rx:=1.8, \Ry:=-2.1, \Rz:=0), v200, z200, Tooldata_7;
MoveJ RelTool (starting_position, 122, 124.9, -442 \Rx:=1.9, \Ry:=-2.1, \Rz:=0), v200, z200, Tooldata_7;
MoveJ RelTool (starting_position, 122, 124.4, -442 \Rx:=2, \Ry:=-2.1, \Rz:=0), v200, z200, Tooldata_7;
MoveJ RelTool (starting_position, 123, 124, -442 \Rx:=2.1, \Ry:=-1.8, \Rz:=0), v200, z200, Tooldata_7;
MoveJ RelTool (starting_position, 123, 123.6, -441 \Rx:=2.2, \Ry:=-1.8, \Rz:=0), v200, z200, Tooldata_7;
MoveJ RelTool (starting_position, 124, 123.2, -441 \Rx:=2.3, \Ry:=-1.8, \Rz:=0), v200, z200, Tooldata_7;
MoveJ RelTool (starting_position, 124, 122.9, -440 \Rx:=2.4, \Ry:=-1.8, \Rz:=0), v200, z200, Tooldata_7;
MoveJ RelTool (starting_position, 125, 122.5, -440 \Rx:=2.6, \Ry:=-1.5, \Rz:=0), v200, z200, Tooldata_7;
MoveJ RelTool (starting_position, 125, 122.3, -440 \Rx:=2.7, \Ry:=-1.5, \Rz:=0), v200, z200, Tooldata_7;
MoveJ RelTool (starting_position, 126, 122, -440 \Rx:=2.9, \Ry:=-1.2, \Rz:=0), v200, z200, Tooldata_7;
MoveJ RelTool (starting_position, 127, 121.7, -439 \Rx:=3.1, \Ry:=-1.2, \Rz:=0), v200, z200, Tooldata_7;
MoveJ RelTool (starting_position, 127, 121.5, -439 \Rx:=3.3, \Ry:=-1.2, \Rz:=0), v200, z200, Tooldata_7;
MoveJ RelTool (starting_position, 128, 121.3, -439 \Rx:=3.6, \Ry:=-0.9, \Rz:=0), v200, z200, Tooldata_7;
MoveJ RelTool (starting_position, 129, 121, -439 \Rx:=3.8, \Ry:=-0.9, \Rz:=0), v200, z200, Tooldata_7;
MoveJ RelTool (starting_position, 130, 120.8, -439 \Rx:=4.1, \Ry:=-0.6, \Rz:=0), v200, z200, Tooldata_7;
MoveJ RelTool (starting_position, 130, 120.6, -439 \Rx:=4.4, \Ry:=-0.6, \Rz:=0), v200, z200, Tooldata_7;
MoveJ RelTool (starting_position, 131, 120.4, -439 \Rx:=4.7, \Ry:=-0.6, \Rz:=0), v200, z200, Tooldata_7;
MoveJ RelTool (starting_position, 131, 120.2, -439 \Rx:=5, \Ry:=-0.3, \Rz:=0), v200, z200, Tooldata_7;
MoveJ RelTool (starting_position, 132, 120, -439 \Rx:=5.2, \Ry:=-0.3, \Rz:=0), v200, z200, Tooldata_7;
MoveJ RelTool (starting_position, 132, 119.8, -439 \Rx:=5.5, \Ry:=-0.3, \Rz:=0), v200, z200, Tooldata_7;
MoveJ RelTool (starting_position, 132, 119.6, -439 \Rx:=5.7, \Ry:=-0.3, \Rz:=0), v200, z200, Tooldata_7;
MoveJ RelTool (starting_position, 133, 119.4, -439 \Rx:=5.9, \Ry:=-0.3, \Rz:=0), v200, z200, Tooldata_7;
MoveJ RelTool (starting_position, 133, 119.2, -440 \Rx:=6.1, \Ry:=-0, \Rz:=0), v200, z200, Tooldata_7;
MoveJ RelTool (starting_position, 133, 119, -440 \Rx:=6.2, \Ry:=-0, \Rz:=0), v200, z200, Tooldata_7;
MoveJ RelTool (starting_position, 134, 118.8, -440 \Rx:=6.3, \Ry:=-0, \Rz:=0), v200, z200, Tooldata_7;
MoveJ RelTool (starting_position, 134, 118.6, -440 \Rx:=6.3, \Ry:=-0, \Rz:=0), v200, z200, Tooldata_7;
MoveJ RelTool (starting_position, 134, 118.3, -441 \Rx:=6.2, \Ry:=-0, \Rz:=0), v200, z200, Tooldata_7;
MoveJ RelTool (starting_position, 133, 118.1, -441 \Rx:=6.1, \Ry:=-0, \Rz:=0), v200, z200, Tooldata_7;
MoveJ RelTool (starting_position, 133, 117.8, -441 \Rx:=6, \Ry:=-0, \Rz:=0), v200, z200, Tooldata_7;
MoveJ RelTool (starting_position, 133, 117.5, -441 \Rx:=5.9, \Ry:=-0.3, \Rz:=0), v200, z200, Tooldata_7;
MoveJ RelTool (starting_position, 132, 117.2, -441 \Rx:=5.6, \Ry:=-0.3, \Rz:=0), v200, z200, Tooldata_7;
MoveJ RelTool (starting_position, 131, 116.8, -442 \Rx:=5.4, \Ry:=-0.3, \Rz:=0), v200, z200, Tooldata_7;
MoveJ RelTool (starting_position, 131, 116.4, -442 \Rx:=5.1, \Ry:=-0.6, \Rz:=0), v200, z200, Tooldata_7;
MoveJ RelTool (starting_position, 130, 116, -442 \Rx:=4.8, \Ry:=-0.6, \Rz:=0), v200, z200, Tooldata_7;
MoveJ RelTool (starting_position, 130, 115.6, -442 \Rx:=4.5, \Ry:=-0.6, \Rz:=0), v200, z200, Tooldata_7;
MoveJ RelTool (starting_position, 129, 115.2, -442 \Rx:=4.2, \Ry:=-0.9, \Rz:=0), v200, z200, Tooldata_7;
MoveJ RelTool (starting_position, 128, 114.7, -442 \Rx:=3.8, \Ry:=-0.9, \Rz:=0), v200, z200, Tooldata_7;
MoveJ RelTool (starting_position, 127, 114.1, -442 \Rx:=3.5, \Ry:=-1.2, \Rz:=0), v200, z200, Tooldata_7;
MoveJ RelTool (starting_position, 127, 113.6, -442 \Rx:=3.2, \Ry:=-1.2, \Rz:=0), v200, z200, Tooldata_7;
MoveJ RelTool (starting_position, 126, 113, -441 \Rx:=2.9, \Ry:=-1.5, \Rz:=0), v200, z200, Tooldata_7;
MoveJ RelTool (starting_position, 125, 112.4, -441 \Rx:=2.6, \Ry:=-1.5, \Rz:=0), v200, z200, Tooldata_7;
MoveJ RelTool (starting_position, 124, 111.8, -441 \Rx:=2.3, \Ry:=-1.5, \Rz:=0), v200, z200, Tooldata_7;
MoveJ RelTool (starting_position, 124, 111.2, -441 \Rx:=2, \Ry:=-1.8, \Rz:=0), v200, z200, Tooldata_7;
MoveJ RelTool (starting_position, 123, 110.5, -440 \Rx:=1.7, \Ry:=-1.8, \Rz:=0), v200, z200, Tooldata_7;
MoveJ RelTool (starting_position, 122, 109.8, -440 \Rx:=1.4, \Ry:=-2.1, \Rz:=0), v200, z200, Tooldata_7;
MoveJ RelTool (starting_position, 122, 109.1, -440 \Rx:=1.2, \Ry:=-2.1, \Rz:=0), v200, z200, Tooldata_7;
MoveJ RelTool (starting_position, 121, 108.4, -439 \Rx:=1.1, \Ry:=-2.1, \Rz:=0), v200, z200, Tooldata_7;
MoveJ RelTool (starting_position, 121, 107.6, -439 \Rx:=0.9, \Ry:=-2.1, \Rz:=0), v200, z200, Tooldata_7;
MoveJ RelTool (starting_position, 120, 106.9, -439 \Rx:=0.8, \Ry:=-2.4, \Rz:=0), v200, z200, Tooldata_7;
MoveJ RelTool (starting_position, 120, 106.2, -438 \Rx:=0.7, \Ry:=-2.4, \Rz:=0), v200, z200, Tooldata_7;
MoveJ RelTool (starting_position, 119, 105.4, -438 \Rx:=0.6, \Ry:=-2.4, \Rz:=0), v200, z200, Tooldata_7;
MoveJ RelTool (starting_position, 119, 104.6, -438 \Rx:=0.6, \Ry:=-2.7, \Rz:=0), v200, z200, Tooldata_7;
MoveJ RelTool (starting_position, 119, 103.9, -437 \Rx:=0.7, \Ry:=-2.7, \Rz:=0), v200, z200, Tooldata_7;
MoveJ RelTool (starting_position, 118, 103.1, -437 \Rx:=0.7, \Ry:=-2.7, \Rz:=0), v200, z200, Tooldata_7;
MoveJ RelTool (starting_position, 118, 102.4, -437 \Rx:=0.9, \Ry:=-2.7, \Rz:=0), v200, z200, Tooldata_7;
MoveJ RelTool (starting_position, 118, 101.7, -436 \Rx:=1.1, \Ry:=-2.7, \Rz:=0), v200, z200, Tooldata_7;
MoveJ RelTool (starting_position, 118, 100.9, -436 \Rx:=1.4, \Ry:=-2.7, \Rz:=0), v200, z200, Tooldata_7;
MoveJ RelTool (starting_position, 117, 100.2, -435 \Rx:=1.7, \Ry:=-2.7, \Rz:=0), v200, z200, Tooldata_7;
MoveJ RelTool (starting_position, 117, 99.5, -435 \Rx:=2.1, \Ry:=-3, \Rz:=0), v200, z200, Tooldata_7;
MoveJ RelTool (starting_position, 117, 98.9, -435 \Rx:=2.5, \Ry:=-3, \Rz:=0), v200, z200, Tooldata_7;
MoveJ RelTool (starting_position, 117, 98.2, -435 \Rx:=3, \Ry:=-3, \Rz:=0), v200, z200, Tooldata_7;
MoveJ RelTool (starting_position, 116, 97.6, -434 \Rx:=3.5, \Ry:=-3, \Rz:=0), v200, z200, Tooldata_7;
MoveJ RelTool (starting_position, 116, 97, -434 \Rx:=4.1, \Ry:=-3, \Rz:=0), v200, z200, Tooldata_7;
MoveJ RelTool (starting_position, 116, 96.4, -434 \Rx:=4.7, \Ry:=-3, \Rz:=0), v200, z200, Tooldata_7;
MoveJ RelTool (starting_position, 116, 95.9, -433 \Rx:=5.3, \Ry:=-3, \Rz:=0), v200, z200, Tooldata_7;
MoveJ RelTool (starting_position, 116, 95.4, -433 \Rx:=6, \Ry:=-3, \Rz:=0), v200, z200, Tooldata_7;
MoveJ RelTool (starting_position, 116, 94.9, -433 \Rx:=6.6, \Ry:=-3, \Rz:=0), v200, z200, Tooldata_7;
MoveJ RelTool (starting_position, 116, 94.4, -432 \Rx:=7.2, \Ry:=-3, \Rz:=0), v200, z200, Tooldata_7;
MoveJ RelTool (starting_position, 116, 94, -432 \Rx:=7.9, \Ry:=-3, \Rz:=0), v200, z200, Tooldata_7;
MoveJ RelTool (starting_position, 116, 93.6, -432 \Rx:=8.5, \Ry:=-3, \Rz:=0), v200, z200, Tooldata_7;
MoveJ RelTool (starting_position, 116, 93.2, -432 \Rx:=9.1, \Ry:=-3, \Rz:=0), v200, z200, Tooldata_7;
MoveJ RelTool (starting_position, 116, 92.9, -431 \Rx:=9.7, \Ry:=-3, \Rz:=0), v200, z200, Tooldata_7;
MoveJ RelTool (starting_position, 116, 92.5, -431 \Rx:=10.2, \Ry:=-3, \Rz:=0), v200, z200, Tooldata_7;
MoveJ RelTool (starting_position, 116, 92.3, -431 \Rx:=10.7, \Ry:=-3, \Rz:=0), v200, z200, Tooldata_7;
MoveJ RelTool (starting_position, 116, 92, -430 \Rx:=11.1, \Ry:=-3, \Rz:=0), v200, z200, Tooldata_7;
MoveJ RelTool (starting_position, 116, 91.7, -430 \Rx:=11.4, \Ry:=-3, \Rz:=0), v200, z200, Tooldata_7;
MoveJ RelTool (starting_position, 116, 91.4, -430 \Rx:=11.6, \Ry:=-3, \Rz:=0), v200, z200, Tooldata_7;
MoveJ RelTool (starting_position, 115, 91.2, -430 \Rx:=11.7, \Ry:=-3.3, \Rz:=0), v200, z200, Tooldata_7;
MoveJ RelTool (starting_position, 115, 90.9, -429 \Rx:=11.8, \Ry:=-3.3, \Rz:=0), v200, z200, Tooldata_7;
MoveJ RelTool (starting_position, 115, 90.7, -429 \Rx:=11.7, \Ry:=-3.3, \Rz:=0), v200, z200, Tooldata_7;
MoveJ RelTool (starting_position, 115, 90.5, -429 \Rx:=11.6, \Ry:=-3.3, \Rz:=0), v200, z200, Tooldata_7;
MoveJ RelTool (starting_position, 115, 90.3, -429 \Rx:=11.4, \Ry:=-3.3, \Rz:=0), v200, z200, Tooldata_7;
MoveJ RelTool (starting_position, 115, 90, -428 \Rx:=11.2, \Ry:=-3.3, \Rz:=0), v200, z200, Tooldata_7;
MoveJ RelTool (starting_position, 115, 89.8, -428 \Rx:=10.9, \Ry:=-3.3, \Rz:=0), v200, z200, Tooldata_7;
MoveJ RelTool (starting_position, 115, 89.6, -428 \Rx:=10.5, \Ry:=-3.3, \Rz:=0), v200, z200, Tooldata_7;
MoveJ RelTool (starting_position, 115, 89.4, -428 \Rx:=10.2, \Ry:=-3.3, \Rz:=0), v200, z200, Tooldata_7;
MoveJ RelTool (starting_position, 114, 89.1, -427 \Rx:=9.7, \Ry:=-3.3, \Rz:=0), v200, z200, Tooldata_7;
MoveJ RelTool (starting_position, 114, 88.9, -427 \Rx:=9.3, \Ry:=-3.3, \Rz:=0), v200, z200, Tooldata_7;
MoveJ RelTool (starting_position, 114, 88.6, -427 \Rx:=8.8, \Ry:=-3.6, \Rz:=0), v200, z200, Tooldata_7;
MoveJ RelTool (starting_position, 113, 88.4, -426 \Rx:=8.3, \Ry:=-3.6, \Rz:=0), v200, z200, Tooldata_7;
MoveJ RelTool (starting_position, 113, 88.1, -426 \Rx:=7.8, \Ry:=-3.6, \Rz:=0), v200, z200, Tooldata_7;
MoveJ RelTool (starting_position, 113, 87.8, -426 \Rx:=7.4, \Ry:=-3.6, \Rz:=0), v200, z200, Tooldata_7;
MoveJ RelTool (starting_position, 113, 87.5, -425 \Rx:=6.9, \Ry:=-3.6, \Rz:=0), v200, z200, Tooldata_7;
MoveJ RelTool (starting_position, 113, 87.2, -425 \Rx:=6.4, \Ry:=-3.6, \Rz:=0), v200, z200, Tooldata_7;
MoveJ RelTool (starting_position, 112, 86.8, -424 \Rx:=6, \Ry:=-3.6, \Rz:=0), v200, z200, Tooldata_7;
MoveJ RelTool (starting_position, 112, 86.4, -424 \Rx:=5.5, \Ry:=-3.9, \Rz:=0), v200, z200, Tooldata_7;
MoveJ RelTool (starting_position, 111, 86, -423 \Rx:=5.1, \Ry:=-3.9, \Rz:=0), v200, z200, Tooldata_7;
MoveJ RelTool (starting_position, 111, 85.6, -423 \Rx:=4.7, \Ry:=-3.9, \Rz:=0), v200, z200, Tooldata_7;
MoveJ RelTool (starting_position, 110, 85.2, -422 \Rx:=4.3, \Ry:=-4.2, \Rz:=0), v200, z200, Tooldata_7;
MoveJ RelTool (starting_position, 109, 84.7, -422 \Rx:=3.9, \Ry:=-4.2, \Rz:=0), v200, z200, Tooldata_7;
MoveJ RelTool (starting_position, 108, 84.1, -421 \Rx:=3.6, \Ry:=-4.5, \Rz:=0), v200, z200, Tooldata_7;
MoveJ RelTool (starting_position, 106, 83.6, -420 \Rx:=3.3, \Ry:=-4.8, \Rz:=0), v200, z200, Tooldata_7;
MoveJ RelTool (starting_position, 105, 83, -420 \Rx:=2.9, \Ry:=-5.1, \Rz:=0), v200, z200, Tooldata_7;
MoveJ RelTool (starting_position, 105, 82.4, -420 \Rx:=2.6, \Ry:=-5.1, \Rz:=0), v200, z200, Tooldata_7;
MoveJ RelTool (starting_position, 104, 81.8, -419 \Rx:=2.4, \Ry:=-5.1, \Rz:=0), v200, z200, Tooldata_7;
MoveJ RelTool (starting_position, 103, 81.2, -419 \Rx:=2.1, \Ry:=-5.4, \Rz:=0), v200, z200, Tooldata_7;
MoveJ RelTool (starting_position, 103, 80.5, -418 \Rx:=1.9, \Ry:=-5.4, \Rz:=0), v200, z200, Tooldata_7;
MoveJ RelTool (starting_position, 102, 79.8, -418 \Rx:=1.6, \Ry:=-5.4, \Rz:=0), v200, z200, Tooldata_7;
MoveJ RelTool (starting_position, 101, 79.1, -418 \Rx:=1.4, \Ry:=-5.7, \Rz:=0), v200, z200, Tooldata_7;
MoveJ RelTool (starting_position, 100, 78.4, -417 \Rx:=1.3, \Ry:=-5.7, \Rz:=0), v200, z200, Tooldata_7;
MoveJ RelTool (starting_position, 99, 77.6, -417 \Rx:=1.1, \Ry:=-6, \Rz:=0), v200, z200, Tooldata_7;
MoveJ RelTool (starting_position, 97, 76.9, -417 \Rx:=1.1, \Ry:=-6.3, \Rz:=0), v200, z200, Tooldata_7;
MoveJ RelTool (starting_position, 95, 76.2, -416 \Rx:=1, \Ry:=-6.6, \Rz:=0), v200, z200, Tooldata_7;
MoveJ RelTool (starting_position, 93, 75.4, -416 \Rx:=1, \Ry:=-6.9, \Rz:=0), v200, z200, Tooldata_7;
MoveJ RelTool (starting_position, 91, 74.6, -416 \Rx:=1, \Ry:=-7.5, \Rz:=0), v200, z200, Tooldata_7;
MoveJ RelTool (starting_position, 88, 73.9, -415 \Rx:=1.1, \Ry:=-7.8, \Rz:=0), v200, z200, Tooldata_7;
MoveJ RelTool (starting_position, 86, 73.1, -415 \Rx:=1.2, \Ry:=-8.4, \Rz:=0), v200, z200, Tooldata_7;
MoveJ RelTool (starting_position, 83, 72.4, -415 \Rx:=1.3, \Ry:=-8.7, \Rz:=0), v200, z200, Tooldata_7;
MoveJ RelTool (starting_position, 81, 71.7, -414 \Rx:=1.5, \Ry:=-9, \Rz:=0), v200, z200, Tooldata_7;
MoveJ RelTool (starting_position, 78, 70.9, -413 \Rx:=1.7, \Ry:=-9.6, \Rz:=0), v200, z200, Tooldata_7;
MoveJ RelTool (starting_position, 75, 70.2, -413 \Rx:=2, \Ry:=-10.2, \Rz:=0), v200, z200, Tooldata_7;
MoveJ RelTool (starting_position, 72, 69.5, -412 \Rx:=2.3, \Ry:=-10.8, \Rz:=0), v200, z200, Tooldata_7;
MoveJ RelTool (starting_position, 70, 68.9, -411 \Rx:=2.7, \Ry:=-11.1, \Rz:=0), v200, z200, Tooldata_7;
MoveJ RelTool (starting_position, 67, 68.2, -410 \Rx:=3.1, \Ry:=-11.7, \Rz:=0), v200, z200, Tooldata_7;
MoveJ RelTool (starting_position, 64, 67.6, -409 \Rx:=3.5, \Ry:=-12, \Rz:=0), v200, z200, Tooldata_7;
MoveJ RelTool (starting_position, 62, 67, -407 \Rx:=4, \Ry:=-12.6, \Rz:=0), v200, z200, Tooldata_7;
MoveJ RelTool (starting_position, 59, 66.4, -406 \Rx:=4.6, \Ry:=-12.9, \Rz:=0), v200, z200, Tooldata_7;
MoveJ RelTool (starting_position, 57, 65.9, -404 \Rx:=5.2, \Ry:=-13.5, \Rz:=0), v200, z200, Tooldata_7;
MoveJ RelTool (starting_position, 55, 65.4, -403 \Rx:=5.8, \Ry:=-13.8, \Rz:=0), v200, z200, Tooldata_7;
MoveJ RelTool (starting_position, 53, 64.9, -401 \Rx:=6.4, \Ry:=-14.1, \Rz:=0), v200, z200, Tooldata_7;
MoveJ RelTool (starting_position, 51, 64.4, -399 \Rx:=7.1, \Ry:=-14.4, \Rz:=0), v200, z200, Tooldata_7;
MoveJ RelTool (starting_position, 49, 64, -397 \Rx:=7.8, \Ry:=-14.7, \Rz:=0), v200, z200, Tooldata_7;
MoveJ RelTool (starting_position, 48, 63.6, -394 \Rx:=8.5, \Ry:=-15, \Rz:=0), v200, z200, Tooldata_7;
MoveJ RelTool (starting_position, 46, 63.2, -392 \Rx:=9.2, \Ry:=-15.3, \Rz:=0), v200, z200, Tooldata_7;
MoveJ RelTool (starting_position, 45, 62.9, -389 \Rx:=9.9, \Ry:=-15.3, \Rz:=0), v200, z200, Tooldata_7;
MoveJ RelTool (starting_position, 45, 62.5, -387 \Rx:=10.5, \Ry:=-15.6, \Rz:=0), v200, z200, Tooldata_7;
MoveJ RelTool (starting_position, 44, 62.3, -384 \Rx:=11.2, \Ry:=-15.6, \Rz:=0), v200, z200, Tooldata_7;
MoveJ RelTool (starting_position, 44, 61.9, -382 \Rx:=11.8, \Ry:=-15.6, \Rz:=0), v200, z200, Tooldata_7;
MoveJ RelTool (starting_position, 44, 61.7, -379 \Rx:=12.3, \Ry:=-15.6, \Rz:=0), v200, z200, Tooldata_7;
MoveJ RelTool (starting_position, 45, 61.4, -376 \Rx:=12.8, \Ry:=-15.3, \Rz:=0), v200, z200, Tooldata_7;
MoveJ RelTool (starting_position, 46, 61.1, -374 \Rx:=13.3, \Ry:=-15.3, \Rz:=0), v200, z200, Tooldata_7;
MoveJ RelTool (starting_position, 47, 60.9, -371 \Rx:=13.7, \Ry:=-15.3, \Rz:=0), v200, z200, Tooldata_7;
MoveJ RelTool (starting_position, 48, 60.6, -368 \Rx:=14.1, \Ry:=-15, \Rz:=0), v200, z200, Tooldata_7;
MoveJ RelTool (starting_position, 50, 60.4, -366 \Rx:=14.4, \Ry:=-14.4, \Rz:=0), v200, z200, Tooldata_7;
MoveJ RelTool (starting_position, 53, 60.1, -363 \Rx:=14.6, \Ry:=-14.1, \Rz:=0), v200, z200, Tooldata_7;
MoveJ RelTool (starting_position, 55, 59.9, -361 \Rx:=14.8, \Ry:=-13.8, \Rz:=0), v200, z200, Tooldata_7;
MoveJ RelTool (starting_position, 58, 59.7, -359 \Rx:=14.9, \Ry:=-13.2, \Rz:=0), v200, z200, Tooldata_7;
MoveJ RelTool (starting_position, 60, 59.4, -356 \Rx:=15, \Ry:=-12.6, \Rz:=0), v200, z200, Tooldata_7;
MoveJ RelTool (starting_position, 63, 59.2, -354 \Rx:=15, \Ry:=-12.3, \Rz:=0), v200, z200, Tooldata_7;
MoveJ RelTool (starting_position, 67, 59, -352 \Rx:=15, \Ry:=-11.7, \Rz:=0), v200, z200, Tooldata_7;
MoveJ RelTool (starting_position, 70, 58.7, -350 \Rx:=14.9, \Ry:=-11.1, \Rz:=0), v200, z200, Tooldata_7;
MoveJ RelTool (starting_position, 74, 58.4, -348 \Rx:=14.8, \Ry:=-10.5, \Rz:=0), v200, z200, Tooldata_7;
MoveJ RelTool (starting_position, 78, 58.1, -347 \Rx:=14.6, \Ry:=-9.6, \Rz:=0), v200, z200, Tooldata_7;
MoveJ RelTool (starting_position, 82, 57.8, -345 \Rx:=14.4, \Ry:=-9, \Rz:=0), v200, z200, Tooldata_7;
MoveJ RelTool (starting_position, 86, 57.5, -344 \Rx:=14.1, \Ry:=-8.1, \Rz:=0), v200, z200, Tooldata_7;
MoveJ RelTool (starting_position, 91, 57.2, -342 \Rx:=13.8, \Ry:=-7.5, \Rz:=0), v200, z200, Tooldata_7;
MoveJ RelTool (starting_position, 95, 56.8, -341 \Rx:=13.5, \Ry:=-6.6, \Rz:=0), v200, z200, Tooldata_7;
MoveJ RelTool (starting_position, 100, 56.4, -340 \Rx:=13.1, \Ry:=-6, \Rz:=0), v200, z200, Tooldata_7;
MoveJ RelTool (starting_position, 104, 56, -339 \Rx:=12.7, \Ry:=-5.1, \Rz:=0), v200, z200, Tooldata_7;
MoveJ RelTool (starting_position, 109, 55.6, -338 \Rx:=12.3, \Ry:=-4.2, \Rz:=0), v200, z200, Tooldata_7;
MoveJ RelTool (starting_position, 113, 55.2, -338 \Rx:=11.8, \Ry:=-3.6, \Rz:=0), v200, z200, Tooldata_7;
MoveJ RelTool (starting_position, 117, 54.7, -337 \Rx:=11.4, \Ry:=-2.7, \Rz:=0), v200, z200, Tooldata_7;
MoveJ RelTool (starting_position, 122, 54.1, -337 \Rx:=10.9, \Ry:=-2.1, \Rz:=0), v200, z200, Tooldata_7;
MoveJ RelTool (starting_position, 126, 53.6, -337 \Rx:=10.4, \Ry:=-1.2, \Rz:=0), v200, z200, Tooldata_7;
MoveJ RelTool (starting_position, 130, 53, -337 \Rx:=10, \Ry:=-0.6, \Rz:=0), v200, z200, Tooldata_7;
MoveJ RelTool (starting_position, 133, 52.4, -338 \Rx:=9.6, \Ry:=0, \Rz:=0), v200, z200, Tooldata_7;
MoveJ RelTool (starting_position, 137, 51.8, -338 \Rx:=9.2, \Ry:=0.6, \Rz:=0), v200, z200, Tooldata_7;
MoveJ RelTool (starting_position, 140, 51.2, -338 \Rx:=8.8, \Ry:=1.2, \Rz:=0), v200, z200, Tooldata_7;
MoveJ RelTool (starting_position, 144, 50.5, -339 \Rx:=8.4, \Ry:=1.8, \Rz:=0), v200, z200, Tooldata_7;
MoveJ RelTool (starting_position, 147, 49.8, -340 \Rx:=8, \Ry:=2.4, \Rz:=0), v200, z200, Tooldata_7;
MoveJ RelTool (starting_position, 150, 49.1, -341 \Rx:=7.6, \Ry:=3, \Rz:=0), v200, z200, Tooldata_7;
MoveJ RelTool (starting_position, 153, 48.4, -341 \Rx:=7.2, \Ry:=3.3, \Rz:=0), v200, z200, Tooldata_7;
MoveJ RelTool (starting_position, 156, 47.6, -342 \Rx:=6.8, \Ry:=3.9, \Rz:=0), v200, z200, Tooldata_7;
MoveJ RelTool (starting_position, 158, 46.9, -343 \Rx:=6.5, \Ry:=4.2, \Rz:=0), v200, z200, Tooldata_7;
MoveJ RelTool (starting_position, 160, 46.2, -344 \Rx:=6.2, \Ry:=4.8, \Rz:=0), v200, z200, Tooldata_7;
MoveJ RelTool (starting_position, 163, 45.4, -345 \Rx:=5.9, \Ry:=5.1, \Rz:=0), v200, z200, Tooldata_7;
MoveJ RelTool (starting_position, 165, 44.6, -346 \Rx:=5.6, \Ry:=5.4, \Rz:=0), v200, z200, Tooldata_7;
MoveJ RelTool (starting_position, 166, 43.9, -347 \Rx:=5.3, \Ry:=5.7, \Rz:=0), v200, z200, Tooldata_7;
MoveJ RelTool (starting_position, 168, 43.1, -348 \Rx:=5, \Ry:=6, \Rz:=0), v200, z200, Tooldata_7;
MoveJ RelTool (starting_position, 169, 42.4, -348 \Rx:=4.6, \Ry:=6.3, \Rz:=0), v200, z200, Tooldata_7;
MoveJ RelTool (starting_position, 170, 41.7, -349 \Rx:=4.3, \Ry:=6.3, \Rz:=0), v200, z200, Tooldata_7;
MoveJ RelTool (starting_position, 171, 40.9, -350 \Rx:=3.9, \Ry:=6.6, \Rz:=0), v200, z200, Tooldata_7;
MoveJ RelTool (starting_position, 171, 40.2, -351 \Rx:=3.6, \Ry:=6.6, \Rz:=0), v200, z200, Tooldata_7;
MoveJ RelTool (starting_position, 172, 39.5, -351 \Rx:=3.2, \Ry:=6.6, \Rz:=0), v200, z200, Tooldata_7;
MoveJ RelTool (starting_position, 172, 38.9, -352 \Rx:=2.8, \Ry:=6.6, \Rz:=0), v200, z200, Tooldata_7;
MoveJ RelTool (starting_position, 172, 38.2, -352 \Rx:=2.5, \Ry:=6.6, \Rz:=0), v200, z200, Tooldata_7;
MoveJ RelTool (starting_position, 172, 37.6, -353 \Rx:=2.1, \Ry:=6.6, \Rz:=0), v200, z200, Tooldata_7;
MoveJ RelTool (starting_position, 172, 37, -353 \Rx:=1.7, \Ry:=6.6, \Rz:=0), v200, z200, Tooldata_7;
MoveJ RelTool (starting_position, 172, 36.4, -354 \Rx:=1.3, \Ry:=6.6, \Rz:=0), v200, z200, Tooldata_7;
MoveJ RelTool (starting_position, 173, 35.9, -354 \Rx:=1, \Ry:=6.6, \Rz:=0), v200, z200, Tooldata_7;
MoveJ RelTool (starting_position, 173, 35.4, -355 \Rx:=0.6, \Ry:=6.9, \Rz:=0), v200, z200, Tooldata_7;
MoveJ RelTool (starting_position, 173, 34.9, -355 \Rx:=0.3, \Ry:=6.9, \Rz:=0), v200, z200, Tooldata_7;
MoveJ RelTool (starting_position, 173, 34.4, -356 \Rx:=-0.1, \Ry:=6.9, \Rz:=0), v200, z200, Tooldata_7;
MoveJ RelTool (starting_position, 173, 34, -356 \Rx:=-0.4, \Ry:=6.9, \Rz:=0), v200, z200, Tooldata_7;
MoveJ RelTool (starting_position, 173, 33.6, -357 \Rx:=-0.6, \Ry:=6.9, \Rz:=0), v200, z200, Tooldata_7;
MoveJ RelTool (starting_position, 173, 33.2, -358 \Rx:=-0.9, \Ry:=6.9, \Rz:=0), v200, z200, Tooldata_7;
MoveJ RelTool (starting_position, 173, 32.9, -358 \Rx:=-1.1, \Ry:=6.9, \Rz:=0), v200, z200, Tooldata_7;
MoveJ RelTool (starting_position, 172, 32.5, -359 \Rx:=-1.3, \Ry:=6.6, \Rz:=0), v200, z200, Tooldata_7;
MoveJ RelTool (starting_position, 172, 32.2, -360 \Rx:=-1.5, \Ry:=6.6, \Rz:=0), v200, z200, Tooldata_7;
MoveJ RelTool (starting_position, 171, 31.8, -360 \Rx:=-1.6, \Ry:=6.6, \Rz:=0), v200, z200, Tooldata_7;
MoveJ RelTool (starting_position, 171, 31.5, -361 \Rx:=-1.7, \Ry:=6.6, \Rz:=0), v200, z200, Tooldata_7;
MoveJ RelTool (starting_position, 170, 31.2, -362 \Rx:=-1.8, \Ry:=6.3, \Rz:=0), v200, z200, Tooldata_7;
MoveJ RelTool (starting_position, 169, 31, -363 \Rx:=-1.8, \Ry:=6, \Rz:=0), v200, z200, Tooldata_7;
MoveJ RelTool (starting_position, 167, 30.7, -364 \Rx:=-1.8, \Ry:=5.7, \Rz:=0), v200, z200, Tooldata_7;
MoveJ RelTool (starting_position, 166, 30.4, -365 \Rx:=-1.8, \Ry:=5.7, \Rz:=0), v200, z200, Tooldata_7;
MoveJ RelTool (starting_position, 165, 30.2, -366 \Rx:=-1.7, \Ry:=5.4, \Rz:=0), v200, z200, Tooldata_7;
MoveJ RelTool (starting_position, 164, 29.9, -367 \Rx:=-1.6, \Ry:=5.4, \Rz:=0), v200, z200, Tooldata_7;
MoveJ RelTool (starting_position, 163, 29.6, -367 \Rx:=-1.5, \Ry:=5.1, \Rz:=0), v200, z200, Tooldata_7;
MoveJ RelTool (starting_position, 161, 29.4, -368 \Rx:=-1.4, \Ry:=4.8, \Rz:=0), v200, z200, Tooldata_7;
MoveJ RelTool (starting_position, 160, 29.1, -369 \Rx:=-1.3, \Ry:=4.5, \Rz:=0), v200, z200, Tooldata_7;
MoveJ RelTool (starting_position, 158, 28.8, -370 \Rx:=-1.3, \Ry:=4.2, \Rz:=0), v200, z200, Tooldata_7;
MoveJ RelTool (starting_position, 156, 28.5, -371 \Rx:=-1.2, \Ry:=3.9, \Rz:=0), v200, z200, Tooldata_7;
MoveJ RelTool (starting_position, 154, 28.2, -371 \Rx:=-1.1, \Ry:=3.6, \Rz:=0), v200, z200, Tooldata_7;
MoveJ RelTool (starting_position, 152, 27.9, -372 \Rx:=-1, \Ry:=3.3, \Rz:=0), v200, z200, Tooldata_7;
MoveJ RelTool (starting_position, 150, 27.6, -372 \Rx:=-1, \Ry:=3, \Rz:=0), v200, z200, Tooldata_7;
MoveJ RelTool (starting_position, 148, 27.2, -373 \Rx:=-1, \Ry:=2.4, \Rz:=0), v200, z200, Tooldata_7;
MoveJ RelTool (starting_position, 146, 26.8, -373 \Rx:=-0.9, \Ry:=2.1, \Rz:=0), v200, z200, Tooldata_7;
MoveJ RelTool (starting_position, 144, 26.4, -374 \Rx:=-0.9, \Ry:=1.8, \Rz:=0), v200, z200, Tooldata_7;
MoveJ RelTool (starting_position, 142, 26, -374 \Rx:=-0.9, \Ry:=1.2, \Rz:=0), v200, z200, Tooldata_7;
MoveJ RelTool (starting_position, 139, 25.6, -374 \Rx:=-0.8, \Ry:=0.9, \Rz:=0), v200, z200, Tooldata_7;
MoveJ RelTool (starting_position, 137, 25.2, -374 \Rx:=-0.8, \Ry:=0.6, \Rz:=0), v200, z200, Tooldata_7;
MoveJ RelTool (starting_position, 136, 24.7, -374 \Rx:=-0.9, \Ry:=0.3, \Rz:=0), v200, z200, Tooldata_7;
MoveJ RelTool (starting_position, 134, 24.1, -374 \Rx:=-0.9, \Ry:=-0, \Rz:=0), v200, z200, Tooldata_7;
MoveJ RelTool (starting_position, 132, 23.6, -373 \Rx:=-1, \Ry:=-0.3, \Rz:=0), v200, z200, Tooldata_7;
MoveJ RelTool (starting_position, 130, 23, -373 \Rx:=-1, \Ry:=-0.6, \Rz:=0), v200, z200, Tooldata_7;
MoveJ RelTool (starting_position, 129, 22.4, -373 \Rx:=-1.1, \Ry:=-0.9, \Rz:=0), v200, z200, Tooldata_7;
MoveJ RelTool (starting_position, 127, 21.8, -372 \Rx:=-1.2, \Ry:=-1.2, \Rz:=0), v200, z200, Tooldata_7;
MoveJ RelTool (starting_position, 126, 21.2, -372 \Rx:=-1.2, \Ry:=-1.5, \Rz:=0), v200, z200, Tooldata_7;
MoveJ RelTool (starting_position, 124, 20.5, -371 \Rx:=-1.3, \Ry:=-1.8, \Rz:=0), v200, z200, Tooldata_7;
MoveJ RelTool (starting_position, 123, 19.8, -371 \Rx:=-1.3, \Ry:=-1.8, \Rz:=0), v200, z200, Tooldata_7;
MoveJ RelTool (starting_position, 123, 19.1, -370 \Rx:=-1.3, \Ry:=-2.1, \Rz:=0), v200, z200, Tooldata_7;
MoveJ RelTool (starting_position, 122, 18.4, -370 \Rx:=-1.4, \Ry:=-2.1, \Rz:=0), v200, z200, Tooldata_7;
MoveJ RelTool (starting_position, 121, 17.6, -369 \Rx:=-1.3, \Ry:=-2.1, \Rz:=0), v200, z200, Tooldata_7;
MoveJ RelTool (starting_position, 121, 16.9, -368 \Rx:=-1.3, \Ry:=-2.1, \Rz:=0), v200, z200, Tooldata_7;
MoveJ RelTool (starting_position, 121, 16.2, -368 \Rx:=-1.3, \Ry:=-2.4, \Rz:=0), v200, z200, Tooldata_7;
MoveJ RelTool (starting_position, 120, 15.4, -367 \Rx:=-1.2, \Ry:=-2.4, \Rz:=0), v200, z200, Tooldata_7;
MoveJ RelTool (starting_position, 120, 14.6, -367 \Rx:=-1.1, \Ry:=-2.4, \Rz:=0), v200, z200, Tooldata_7;
MoveJ RelTool (starting_position, 120, 13.9, -366 \Rx:=-1, \Ry:=-2.4, \Rz:=0), v200, z200, Tooldata_7;
MoveJ RelTool (starting_position, 121, 13.1, -366 \Rx:=-0.9, \Ry:=-2.4, \Rz:=0), v200, z200, Tooldata_7;
MoveJ RelTool (starting_position, 121, 12.4, -365 \Rx:=-0.8, \Ry:=-2.1, \Rz:=0), v200, z200, Tooldata_7;
MoveJ RelTool (starting_position, 122, 11.7, -365 \Rx:=-0.6, \Ry:=-2.1, \Rz:=0), v200, z200, Tooldata_7;
MoveJ RelTool (starting_position, 122, 10.9, -365 \Rx:=-0.4, \Ry:=-2.1, \Rz:=0), v200, z200, Tooldata_7;
MoveJ RelTool (starting_position, 123, 10.2, -364 \Rx:=-0.2, \Ry:=-1.8, \Rz:=0), v200, z200, Tooldata_7;
MoveJ RelTool (starting_position, 124, 9.5, -364 \Rx:=-0, \Ry:=-1.8, \Rz:=0), v200, z200, Tooldata_7;
MoveJ RelTool (starting_position, 124, 8.9, -364 \Rx:=0.2, \Ry:=-1.5, \Rz:=0), v200, z200, Tooldata_7;
MoveJ RelTool (starting_position, 125, 8.2, -363 \Rx:=0.4, \Ry:=-1.5, \Rz:=0), v200, z200, Tooldata_7;
MoveJ RelTool (starting_position, 126, 7.6, -363 \Rx:=0.7, \Ry:=-1.5, \Rz:=0), v200, z200, Tooldata_7;
MoveJ RelTool (starting_position, 126, 7, -363 \Rx:=0.9, \Ry:=-1.2, \Rz:=0), v200, z200, Tooldata_7;
MoveJ RelTool (starting_position, 127, 6.4, -363 \Rx:=1.1, \Ry:=-1.2, \Rz:=0), v200, z200, Tooldata_7;
MoveJ RelTool (starting_position, 128, 5.9, -363 \Rx:=1.3, \Ry:=-0.9, \Rz:=0), v200, z200, Tooldata_7;
MoveJ RelTool (starting_position, 129, 5.4, -363 \Rx:=1.5, \Ry:=-0.9, \Rz:=0), v200, z200, Tooldata_7;
MoveJ RelTool (starting_position, 130, 4.9, -363 \Rx:=1.8, \Ry:=-0.6, \Rz:=0), v200, z200, Tooldata_7;
MoveJ RelTool (starting_position, 131, 4.4, -363 \Rx:=2, \Ry:=-0.6, \Rz:=0), v200, z200, Tooldata_7;
MoveJ RelTool (starting_position, 132, 4, -363 \Rx:=2.3, \Ry:=-0.3, \Rz:=0), v200, z200, Tooldata_7;
MoveJ RelTool (starting_position, 133, 3.6, -363 \Rx:=2.6, \Ry:=-0, \Rz:=0), v200, z200, Tooldata_7;
MoveJ RelTool (starting_position, 134, 3.2, -363 \Rx:=2.9, \Ry:=-0, \Rz:=0), v200, z200, Tooldata_7;
MoveJ RelTool (starting_position, 134, 2.9, -363 \Rx:=3.2, \Ry:=0, \Rz:=0), v200, z200, Tooldata_7;
MoveJ RelTool (starting_position, 135, 2.5, -363 \Rx:=3.5, \Ry:=0.3, \Rz:=0), v200, z200, Tooldata_7;
MoveJ RelTool (starting_position, 135, 2.2, -364 \Rx:=3.8, \Ry:=0.3, \Rz:=0), v200, z200, Tooldata_7;
MoveJ RelTool (starting_position, 136, 1.8, -364 \Rx:=4.1, \Ry:=0.3, \Rz:=0), v200, z200, Tooldata_7;
MoveJ RelTool (starting_position, 136, 1.5, -364 \Rx:=4.5, \Ry:=0.6, \Rz:=0), v200, z200, Tooldata_7;
MoveJ RelTool (starting_position, 137, 1.2, -364 \Rx:=4.8, \Ry:=0.6, \Rz:=0), v200, z200, Tooldata_7;
MoveJ RelTool (starting_position, 137, 1, -365 \Rx:=5, \Ry:=0.6, \Rz:=0), v200, z200, Tooldata_7;
MoveJ RelTool (starting_position, 137, 0.7, -365 \Rx:=5.2, \Ry:=0.6, \Rz:=0), v200, z200, Tooldata_7;
MoveJ RelTool (starting_position, 138, 0.4, -365 \Rx:=5.4, \Ry:=0.6, \Rz:=0), v200, z200, Tooldata_7;
MoveJ RelTool (starting_position, 138, 0.2, -365 \Rx:=5.6, \Ry:=0.6, \Rz:=0), v200, z200, Tooldata_7;
MoveJ RelTool (starting_position, 138, -0.1, -366 \Rx:=5.8, \Ry:=0.9, \Rz:=0), v200, z200, Tooldata_7;
MoveJ RelTool (starting_position, 138, -0.4, -366 \Rx:=5.8, \Ry:=0.9, \Rz:=0), v200, z200, Tooldata_7;
MoveJ RelTool (starting_position, 138, -0.6, -366 \Rx:=5.9, \Ry:=0.9, \Rz:=0), v200, z200, Tooldata_7;
MoveJ RelTool (starting_position, 138, -0.9, -366 \Rx:=5.8, \Ry:=0.6, \Rz:=0), v200, z200, Tooldata_7;
MoveJ RelTool (starting_position, 137, -1.2, -367 \Rx:=5.8, \Ry:=0.6, \Rz:=0), v200, z200, Tooldata_7;
MoveJ RelTool (starting_position, 137, -1.5, -367 \Rx:=5.7, \Ry:=0.6, \Rz:=0), v200, z200, Tooldata_7;
MoveJ RelTool (starting_position, 136, -1.8, -367 \Rx:=5.6, \Ry:=0.3, \Rz:=0), v200, z200, Tooldata_7;
MoveJ RelTool (starting_position, 136, -2.1, -367 \Rx:=5.5, \Ry:=0.3, \Rz:=0), v200, z200, Tooldata_7;
MoveJ RelTool (starting_position, 135, -2.4, -367 \Rx:=5.3, \Ry:=0.3, \Rz:=0), v200, z200, Tooldata_7;
MoveJ RelTool (starting_position, 135, -2.8, -367 \Rx:=5.1, \Ry:=0.3, \Rz:=0), v200, z200, Tooldata_7;
MoveJ RelTool (starting_position, 134, -3.2, -367 \Rx:=4.8, \Ry:=0, \Rz:=0), v200, z200, Tooldata_7;
MoveJ RelTool (starting_position, 133, -3.6, -367 \Rx:=4.6, \Ry:=-0, \Rz:=0), v200, z200, Tooldata_7;
MoveJ RelTool (starting_position, 132, -4, -367 \Rx:=4.4, \Ry:=-0.3, \Rz:=0), v200, z200, Tooldata_7;
MoveJ RelTool (starting_position, 131, -4.4, -367 \Rx:=4.1, \Ry:=-0.6, \Rz:=0), v200, z200, Tooldata_7;
MoveJ RelTool (starting_position, 130, -4.8, -367 \Rx:=3.9, \Ry:=-0.6, \Rz:=0), v200, z200, Tooldata_7;
MoveJ RelTool (starting_position, 130, -5.3, -367 \Rx:=3.7, \Ry:=-0.6, \Rz:=0), v200, z200, Tooldata_7;
MoveJ RelTool (starting_position, 129, -5.9, -367 \Rx:=3.5, \Ry:=-0.9, \Rz:=0), v200, z200, Tooldata_7;
MoveJ RelTool (starting_position, 128, -6.4, -366 \Rx:=3.3, \Ry:=-0.9, \Rz:=0), v200, z200, Tooldata_7;
MoveJ RelTool (starting_position, 127, -7, -366 \Rx:=3.1, \Ry:=-1.2, \Rz:=0), v200, z200, Tooldata_7;
MoveJ RelTool (starting_position, 126, -7.6, -366 \Rx:=3, \Ry:=-1.2, \Rz:=0), v200, z200, Tooldata_7;
MoveJ RelTool (starting_position, 126, -8.2, -366 \Rx:=2.9, \Ry:=-1.5, \Rz:=0), v200, z200, Tooldata_7;
MoveJ RelTool (starting_position, 125, -8.8, -365 \Rx:=2.7, \Ry:=-1.5, \Rz:=0), v200, z200, Tooldata_7;
MoveJ RelTool (starting_position, 124, -9.5, -365 \Rx:=2.6, \Ry:=-1.8, \Rz:=0), v200, z200, Tooldata_7;
MoveJ RelTool (starting_position, 123, -10.2, -365 \Rx:=2.5, \Ry:=-1.8, \Rz:=0), v200, z200, Tooldata_7;
